ACTION TEST_CASE_2_EXEC:
                        IF vTestCases[1].state = utTestCaseStates.ut_RUNNING THEN
	(*Run the test case*)
	IF NOT assertNotEqual_STRING(vTestCase2_act, vTestCase2_xp) THEN
		vTestCases[1].state := utTestCaseStates.ut_PASSED;
		vTestCases[1].msg := 'Passed parameters were equal and function returned FALSE -> PASS';
	ELSE
		vTestCases[1].state := utTestCaseStates.ut_FAILED;
		vTestCases[1].msg := 'Passed parameters were equal and function returned TRUE -> FAIL';
	END_IF
END_IF
                      
END_ACTION
END_PROGRAM

PROGRAM test_assertNotEqual_TIME_OF_DAY
  VAR
    vTestCases : ARRAY[0..20] OF utTestCase;  (* Definition of all test cases for this POU *)
    testRunner : utTestSuite;  (* Test Suite fb instance to run the tests *)
    vRunAll : BOOL;  (* Manual command to run all tests for this POU *)
    vResetAll : BOOL;  (* Manual command to reset all tests for this POU *)
    vTestCase1_act : TOD;  (* Test data 1 of test case 1 *)
    vTestCase1_xp : TOD;  (* Test data 2 of test case 1 *)
    vTestCase2_act : TOD;  (* Test data 1 of test case 2 *)
    vTestCase2_xp : TOD;  (* Test data 2 of test case 2 *)
  END_VAR

                    (*Run the test cases*)
TEST_CASE_1_SETUP();
TEST_CASE_1_EXEC();

TEST_CASE_2_SETUP();
TEST_CASE_2_EXEC();

(*Instantiate the test runner*)
testRunner(
	Id := 48,
	Name := 'assertNotEqual_TIME_OF_DAY',
    RunTests := GVL.RunAll OR vRunAll,
	ResetTests := GVL.ResetAll OR vResetAll,
	TestCases:=vTestCases);

(*Report the results to the collection global*)
GVL.Results[testRunner.Id] := testRunner.Summary;
                  

ACTION TEST_CASE_2_EXEC:
                        IF vTestCases[1].state = utTestCaseStates.ut_RUNNING THEN
	(*Run the test case*)
	IF NOT assertNotEqual_TIME_OF_DAY(vTestCase2_act, vTestCase2_xp) THEN
		vTestCases[1].state := utTestCaseStates.ut_PASSED;
		vTestCases[1].msg := 'Passed parameters were equal and function returned FALSE -> PASS';
	ELSE
		vTestCases[1].state := utTestCaseStates.ut_FAILED;
		vTestCases[1].msg := 'Passed parameters were equal and function returned TRUE -> FAIL';
	END_IF
END_IF
                      
END_ACTION

ACTION TEST_CASE_1_SETUP:
                        IF vTestCases[0].state = utTestCaseStates.ut_SETUP THEN
	(*Setup the test case information*)
	vTestCases[0].id := 1;
	vTestCases[0].desc[0] := 'RETURNS TRUE WHEN PARAMETERS NOT EQUAL';
    vTestCases[0].desc[1] := 'Tests if the function returns True if the passed in parameters do not hold the same value';
	vTestCases[0].desc[2] := 'PASS IF: Return value is TRUE';
	
	(*Setup needed variables*)
	vTestCase1_act := REAL_TO_TOD(115.4);
	vTestCase1_xp := REAL_TO_TOD(-85.4);
END_IF
                      
END_ACTION

ACTION TEST_CASE_1_EXEC:
                        IF vTestCases[0].state = utTestCaseStates.ut_RUNNING THEN
	(*Run the test case*)
	IF assertNotEqual_TIME_OF_DAY(vTestCase1_act, vTestCase1_xp) THEN
		vTestCases[0].state := utTestCaseStates.ut_PASSED;
		vTestCases[0].msg := 'Passed parameters were not equal and function returned TRUE -> PASS';
	ELSE
		vTestCases[0].state := utTestCaseStates.ut_FAILED;
		vTestCases[0].msg := 'Passed parameters were not equal and function returned FALSE -> FAIL';
	END_IF
END_IF
                      
END_ACTION

ACTION TEST_CASE_2_SETUP:
                        IF vTestCases[1].state = utTestCaseStates.ut_SETUP THEN
	(*Setup the test case information*)
	vTestCases[1].id := 2;
	vTestCases[1].desc[0] := 'RETURNS FALSE WHEN PARAMETERS EQUAL';
    vTestCases[1].desc[1] := 'Tests if the function returns False if the passed in parameters hold the same value';
	vTestCases[1].desc[2] := 'PASS IF: Return value is FALSE';
	
	(*Setup needed variables*)
	vTestCase2_act := REAL_TO_TOD(115.4);
	vTestCase2_xp := REAL_TO_TOD(115.4);
END_IF
                      
END_ACTION
END_PROGRAM

PROGRAM test_assertGreater_UDINT
  VAR
    vTestCases : ARRAY[0..20] OF utTestCase;  (* Definition of all test cases for this POU *)
    testRunner : utTestSuite;  (* Test Suite fb instance to run the tests *)
    vRunAll : BOOL;  (* Manual command to run all tests for this POU *)
    vResetAll : BOOL;  (* Manual command to reset all tests for this POU *)
    vTestCase1_act : UDINT;  (* Test data 1 of test case 1 *)
    vTestCase1_xp : UDINT;  (* Test data 2 of test case 1 *)
    vTestCase2_act : UDINT;  (* Test data 1 of test case 2 *)
    vTestCase2_xp : UDINT;  (* Test data 2 of test case 2 *)
  END_VAR

                    (*Run the test cases*)
TEST_CASE_1_SETUP();
TEST_CASE_1_EXEC();

TEST_CASE_2_SETUP();
TEST_CASE_2_EXEC();

(*Instantiate the test runner*)
testRunner(
	Id := 59,
	Name := 'assertGreater_UDINT',
    RunTests := GVL.RunAll OR vRunAll,
	ResetTests := GVL.ResetAll OR vResetAll,
	TestCases:=vTestCases);

(*Report the results to the collection global*)
GVL.Results[testRunner.Id] := testRunner.Summary;
                  

ACTION TEST_CASE_1_SETUP:
                        IF vTestCases[0].state = utTestCaseStates.ut_SETUP THEN
	(*Setup the test case information*)
	vTestCases[0].id := 1;
	vTestCases[0].desc[0] := 'RETURNS TRUE WHEN PARAMETER ACT GREATER THAN XP';
    vTestCases[0].desc[1] := 'Tests if the function returns True if the parameter act is greater than parameter xp';
	vTestCases[0].desc[2] := 'PASS IF: Return value is TRUE';
	
	(*Setup needed variables*)
	vTestCase1_act := REAL_TO_UDINT(115.4);
	vTestCase1_xp := REAL_TO_UDINT(85.4);
END_IF
                      
END_ACTION

ACTION TEST_CASE_1_EXEC:
                        IF vTestCases[0].state = utTestCaseStates.ut_RUNNING THEN
	(*Run the test case*)
	IF assertGreater_UDINT(vTestCase1_act, vTestCase1_xp) THEN
		vTestCases[0].state := utTestCaseStates.ut_PASSED;
		vTestCases[0].msg := 'Parameter act was greater than xp and function returned TRUE -> PASS';
	ELSE
		vTestCases[0].state := utTestCaseStates.ut_FAILED;
		vTestCases[0].msg := 'Parameter act was greater than xp and function returned FALSE -> FAIL';
	END_IF
END_IF
                      
END_ACTION

ACTION TEST_CASE_2_SETUP:
                        IF vTestCases[1].state = utTestCaseStates.ut_SETUP THEN
	(*Setup the test case information*)
	vTestCases[1].id := 2;
    vTestCases[1].desc[0] := 'RETURNS FALSE WHEN PARAMETER ACT LESS THAN XP';
    vTestCases[1].desc[1] := 'Tests if the function returns False if the parameter act is less than parameter xp';
	vTestCases[1].desc[2] := 'PASS IF: Return value is FALSE';
	
	(*Setup needed variables*)
	vTestCase2_act := REAL_TO_UDINT(8.4);
	vTestCase2_xp := REAL_TO_UDINT(85.4);
END_IF
                      
END_ACTION

ACTION TEST_CASE_2_EXEC:
                        IF vTestCases[1].state = utTestCaseStates.ut_RUNNING THEN
	(*Run the test case*)
	IF NOT assertGreater_UDINT(vTestCase2_act, vTestCase2_xp) THEN
		vTestCases[1].state := utTestCaseStates.ut_PASSED;
		vTestCases[1].msg := 'Parameter act was less than xp and function returned FALSE -> PASS';
	ELSE
		vTestCases[1].state := utTestCaseStates.ut_FAILED;
		vTestCases[1].msg := 'Parameter act was less than xp and function returned TRUE -> FAIL';
	END_IF
END_IF
                      
END_ACTION
END_PROGRAM

PROGRAM test_assertNotEqual_LTIME_OF_DAY
  VAR
    vTestCases : ARRAY[0..20] OF utTestCase;  (* Definition of all test cases for this POU *)
    testRunner : utTestSuite;  (* Test Suite fb instance to run the tests *)
    vRunAll : BOOL;  (* Manual command to run all tests for this POU *)
    vResetAll : BOOL;  (* Manual command to reset all tests for this POU *)
    vTestCase1_act : LTIME_OF_DAY;  (* Test data 1 of test case 1 *)
    vTestCase1_xp : LTIME_OF_DAY;  (* Test data 2 of test case 1 *)
    vTestCase2_act : LTIME_OF_DAY;  (* Test data 1 of test case 2 *)
    vTestCase2_xp : LTIME_OF_DAY;  (* Test data 2 of test case 2 *)
  END_VAR

                    (*Run the test cases*)
TEST_CASE_1_SETUP();
TEST_CASE_1_EXEC();

TEST_CASE_2_SETUP();
TEST_CASE_2_EXEC();

(*Instantiate the test runner*)
testRunner(
	Id := 49,
	Name := 'assertNotEqual_LTIME_OF_DAY',
    RunTests := GVL.RunAll OR vRunAll,
	ResetTests := GVL.ResetAll OR vResetAll,
	TestCases:=vTestCases);

(*Report the results to the collection global*)
GVL.Results[testRunner.Id] := testRunner.Summary;
                  

ACTION TEST_CASE_1_SETUP:
                        IF vTestCases[0].state = utTestCaseStates.ut_SETUP THEN
	(*Setup the test case information*)
	vTestCases[0].id := 1;
	vTestCases[0].desc[0] := 'RETURNS TRUE WHEN PARAMETERS NOT EQUAL';
    vTestCases[0].desc[1] := 'Tests if the function returns True if the passed in parameters do not hold the same value';
	vTestCases[0].desc[2] := 'PASS IF: Return value is TRUE';
	
	(*Setup needed variables*)
	vTestCase1_act := REAL_TO_LTOD(115.4);
	vTestCase1_xp := REAL_TO_LTOD(-85.4);
END_IF
                      
END_ACTION

ACTION TEST_CASE_1_EXEC:
                        IF vTestCases[0].state = utTestCaseStates.ut_RUNNING THEN
	(*Run the test case*)
	IF assertNotEqual_LTIME_OF_DAY(vTestCase1_act, vTestCase1_xp) THEN
		vTestCases[0].state := utTestCaseStates.ut_PASSED;
		vTestCases[0].msg := 'Passed parameters were not equal and function returned TRUE -> PASS';
	ELSE
		vTestCases[0].state := utTestCaseStates.ut_FAILED;
		vTestCases[0].msg := 'Passed parameters were not equal and function returned FALSE -> FAIL';
	END_IF
END_IF
                      
END_ACTION

ACTION TEST_CASE_2_SETUP:
                        IF vTestCases[1].state = utTestCaseStates.ut_SETUP THEN
	(*Setup the test case information*)
	vTestCases[1].id := 2;
	vTestCases[1].desc[0] := 'RETURNS FALSE WHEN PARAMETERS EQUAL';
    vTestCases[1].desc[1] := 'Tests if the function returns False if the passed in parameters hold the same value';
	vTestCases[1].desc[2] := 'PASS IF: Return value is FALSE';
	
	(*Setup needed variables*)
	vTestCase2_act := REAL_TO_LTOD(115.4);
	vTestCase2_xp := REAL_TO_LTOD(115.4);
END_IF
                      
END_ACTION

ACTION TEST_CASE_2_EXEC:
                        IF vTestCases[1].state = utTestCaseStates.ut_RUNNING THEN
	(*Run the test case*)
	IF NOT assertNotEqual_LTIME_OF_DAY(vTestCase2_act, vTestCase2_xp) THEN
		vTestCases[1].state := utTestCaseStates.ut_PASSED;
		vTestCases[1].msg := 'Passed parameters were equal and function returned FALSE -> PASS';
	ELSE
		vTestCases[1].state := utTestCaseStates.ut_FAILED;
		vTestCases[1].msg := 'Passed parameters were equal and function returned TRUE -> FAIL';
	END_IF
END_IF
                      
END_ACTION
END_PROGRAM

PROGRAM test_assertGreater_BYTE
  VAR
    vTestCases : ARRAY[0..20] OF utTestCase;  (* Definition of all test cases for this POU *)
    testRunner : utTestSuite;  (* Test Suite fb instance to run the tests *)
    vRunAll : BOOL;  (* Manual command to run all tests for this POU *)
    vResetAll : BOOL;  (* Manual command to reset all tests for this POU *)
    vTestCase1_act : BYTE;  (* Test data 1 of test case 1 *)
    vTestCase1_xp : BYTE;  (* Test data 2 of test case 1 *)
    vTestCase2_act : BYTE;  (* Test data 1 of test case 2 *)
    vTestCase2_xp : BYTE;  (* Test data 2 of test case 2 *)
  END_VAR

                    (*Run the test cases*)
TEST_CASE_1_SETUP();
TEST_CASE_1_EXEC();

TEST_CASE_2_SETUP();
TEST_CASE_2_EXEC();

(*Instantiate the test runner*)
testRunner(
	Id := 50,
	Name := 'assertGreater_BYTE',
    RunTests := GVL.RunAll OR vRunAll,
	ResetTests := GVL.ResetAll OR vResetAll,
	TestCases:=vTestCases);

(*Report the results to the collection global*)
GVL.Results[testRunner.Id] := testRunner.Summary;
                  

ACTION TEST_CASE_1_SETUP:
                        IF vTestCases[0].state = utTestCaseStates.ut_SETUP THEN
	(*Setup the test case information*)
	vTestCases[0].id := 1;
	vTestCases[0].desc[0] := 'RETURNS TRUE WHEN PARAMETER ACT GREATER THAN XP';
    vTestCases[0].desc[1] := 'Tests if the function returns True if the parameter act is greater than parameter xp';
	vTestCases[0].desc[2] := 'PASS IF: Return value is TRUE';
	
	(*Setup needed variables*)
	vTestCase1_act := REAL_TO_BYTE(115.4);
	vTestCase1_xp := REAL_TO_BYTE(85.4);
END_IF
                      
END_ACTION

ACTION TEST_CASE_1_EXEC:
                        IF vTestCases[0].state = utTestCaseStates.ut_RUNNING THEN
	(*Run the test case*)
	IF assertGreater_BYTE(vTestCase1_act, vTestCase1_xp) THEN
		vTestCases[0].state := utTestCaseStates.ut_PASSED;
		vTestCases[0].msg := 'Parameter act was greater than xp and function returned TRUE -> PASS';
	ELSE
		vTestCases[0].state := utTestCaseStates.ut_FAILED;
		vTestCases[0].msg := 'Parameter act was greater than xp and function returned FALSE -> FAIL';
	END_IF
END_IF
                      
END_ACTION

ACTION TEST_CASE_2_SETUP:
                        IF vTestCases[1].state = utTestCaseStates.ut_SETUP THEN
	(*Setup the test case information*)
	vTestCases[1].id := 2;
    vTestCases[1].desc[0] := 'RETURNS FALSE WHEN PARAMETER ACT LESS THAN XP';
    vTestCases[1].desc[1] := 'Tests if the function returns False if the parameter act is less than parameter xp';
	vTestCases[1].desc[2] := 'PASS IF: Return value is FALSE';
	
	(*Setup needed variables*)
	vTestCase2_act := REAL_TO_BYTE(8.4);
	vTestCase2_xp := REAL_TO_BYTE(85.4);
END_IF
                      
END_ACTION

ACTION TEST_CASE_2_EXEC:
                        IF vTestCases[1].state = utTestCaseStates.ut_RUNNING THEN
	(*Run the test case*)
	IF NOT assertGreater_BYTE(vTestCase2_act, vTestCase2_xp) THEN
		vTestCases[1].state := utTestCaseStates.ut_PASSED;
		vTestCases[1].msg := 'Parameter act was less than xp and function returned FALSE -> PASS';
	ELSE
		vTestCases[1].state := utTestCaseStates.ut_FAILED;
		vTestCases[1].msg := 'Parameter act was less than xp and function returned TRUE -> FAIL';
	END_IF
END_IF
                      
END_ACTION
END_PROGRAM

PROGRAM test_assertNotEqual_WSTRING
  VAR
    vTestCases : ARRAY[0..20] OF utTestCase;  (* Definition of all test cases for this POU *)
    testRunner : utTestSuite;  (* Test Suite fb instance to run the tests *)
    vRunAll : BOOL;  (* Manual command to run all tests for this POU *)
    vResetAll : BOOL;  (* Manual command to reset all tests for this POU *)
    vTestCase1_act : WSTRING;  (* Test data 1 of test case 1 *)
    vTestCase1_xp : WSTRING;  (* Test data 2 of test case 1 *)
    vTestCase2_act : WSTRING;  (* Test data 1 of test case 2 *)
    vTestCase2_xp : WSTRING;  (* Test data 2 of test case 2 *)
  END_VAR

                    (*Run the test cases*)
TEST_CASE_1_SETUP();
TEST_CASE_1_EXEC();

TEST_CASE_2_SETUP();
TEST_CASE_2_EXEC();

(*Instantiate the test runner*)
testRunner(
	Id := 41,
	Name := 'assertNotEqual_WSTRING',
    RunTests := GVL.RunAll OR vRunAll,
	ResetTests := GVL.ResetAll OR vResetAll,
	TestCases:=vTestCases);

(*Report the results to the collection global*)
GVL.Results[testRunner.Id] := testRunner.Summary;
                  

ACTION TEST_CASE_2_EXEC:
                        IF vTestCases[1].state = utTestCaseStates.ut_RUNNING THEN
	(*Run the test case*)
	IF NOT assertNotEqual_WSTRING(vTestCase2_act, vTestCase2_xp) THEN
		vTestCases[1].state := utTestCaseStates.ut_PASSED;
		vTestCases[1].msg := 'Passed parameters were equal and function returned FALSE -> PASS';
	ELSE
		vTestCases[1].state := utTestCaseStates.ut_FAILED;
		vTestCases[1].msg := 'Passed parameters were equal and function returned TRUE -> FAIL';
	END_IF
END_IF
                      
END_ACTION

ACTION TEST_CASE_1_SETUP:
                        IF vTestCases[0].state = utTestCaseStates.ut_SETUP THEN
	(*Setup the test case information*)
	vTestCases[0].id := 1;
	vTestCases[0].desc[0] := 'RETURNS TRUE WHEN PARAMETERS NOT EQUAL';
    vTestCases[0].desc[1] := 'Tests if the function returns True if the passed in parameters do not hold the same value';
	vTestCases[0].desc[2] := 'PASS IF: Return value is TRUE';
	
	(*Setup needed variables*)
	vTestCase1_act := REAL_TO_WSTRING(115.4);
	vTestCase1_xp := REAL_TO_WSTRING(-85.4);
END_IF
                      
END_ACTION

ACTION TEST_CASE_1_EXEC:
                        IF vTestCases[0].state = utTestCaseStates.ut_RUNNING THEN
	(*Run the test case*)
	IF assertNotEqual_WSTRING(vTestCase1_act, vTestCase1_xp) THEN
		vTestCases[0].state := utTestCaseStates.ut_PASSED;
		vTestCases[0].msg := 'Passed parameters were not equal and function returned TRUE -> PASS';
	ELSE
		vTestCases[0].state := utTestCaseStates.ut_FAILED;
		vTestCases[0].msg := 'Passed parameters were not equal and function returned FALSE -> FAIL';
	END_IF
END_IF
                      
END_ACTION

ACTION TEST_CASE_2_SETUP:
                        IF vTestCases[1].state = utTestCaseStates.ut_SETUP THEN
	(*Setup the test case information*)
	vTestCases[1].id := 2;
	vTestCases[1].desc[0] := 'RETURNS FALSE WHEN PARAMETERS EQUAL';
    vTestCases[1].desc[1] := 'Tests if the function returns False if the passed in parameters hold the same value';
	vTestCases[1].desc[2] := 'PASS IF: Return value is FALSE';
	
	(*Setup needed variables*)
	vTestCase2_act := REAL_TO_WSTRING(115.4);
	vTestCase2_xp := REAL_TO_WSTRING(115.4);
END_IF
                      
END_ACTION
END_PROGRAM

PROGRAM test_assertNotEqual_DWORD
  VAR
    vTestCases : ARRAY[0..20] OF utTestCase;  (* Definition of all test cases for this POU *)
    testRunner : utTestSuite;  (* Test Suite fb instance to run the tests *)
    vRunAll : BOOL;  (* Manual command to run all tests for this POU *)
    vResetAll : BOOL;  (* Manual command to reset all tests for this POU *)
    vTestCase1_act : DWORD;  (* Test data 1 of test case 1 *)
    vTestCase1_xp : DWORD;  (* Test data 2 of test case 1 *)
    vTestCase2_act : DWORD;  (* Test data 1 of test case 2 *)
    vTestCase2_xp : DWORD;  (* Test data 2 of test case 2 *)
  END_VAR

                    (*Run the test cases*)
TEST_CASE_1_SETUP();
TEST_CASE_1_EXEC();

TEST_CASE_2_SETUP();
TEST_CASE_2_EXEC();

(*Instantiate the test runner*)
testRunner(
	Id := 28,
	Name := 'assertNotEqual_DWORD',
    RunTests := GVL.RunAll OR vRunAll,
	ResetTests := GVL.ResetAll OR vResetAll,
	TestCases:=vTestCases);

(*Report the results to the collection global*)
GVL.Results[testRunner.Id] := testRunner.Summary;
                  

ACTION TEST_CASE_1_SETUP:
                        IF vTestCases[0].state = utTestCaseStates.ut_SETUP THEN
	(*Setup the test case information*)
	vTestCases[0].id := 1;
	vTestCases[0].desc[0] := 'RETURNS TRUE WHEN PARAMETERS NOT EQUAL';
    vTestCases[0].desc[1] := 'Tests if the function returns True if the passed in parameters do not hold the same value';
	vTestCases[0].desc[2] := 'PASS IF: Return value is TRUE';
	
	(*Setup needed variables*)
	vTestCase1_act := REAL_TO_DWORD(115.4);
	vTestCase1_xp := REAL_TO_DWORD(-85.4);
END_IF
                      
END_ACTION

ACTION TEST_CASE_1_EXEC:
                        IF vTestCases[0].state = utTestCaseStates.ut_RUNNING THEN
	(*Run the test case*)
	IF assertNotEqual_DWORD(vTestCase1_act, vTestCase1_xp) THEN
		vTestCases[0].state := utTestCaseStates.ut_PASSED;
		vTestCases[0].msg := 'Passed parameters were not equal and function returned TRUE -> PASS';
	ELSE
		vTestCases[0].state := utTestCaseStates.ut_FAILED;
		vTestCases[0].msg := 'Passed parameters were not equal and function returned FALSE -> FAIL';
	END_IF
END_IF
                      
END_ACTION

ACTION TEST_CASE_2_SETUP:
                        IF vTestCases[1].state = utTestCaseStates.ut_SETUP THEN
	(*Setup the test case information*)
	vTestCases[1].id := 2;
	vTestCases[1].desc[0] := 'RETURNS FALSE WHEN PARAMETERS EQUAL';
    vTestCases[1].desc[1] := 'Tests if the function returns False if the passed in parameters hold the same value';
	vTestCases[1].desc[2] := 'PASS IF: Return value is FALSE';
	
	(*Setup needed variables*)
	vTestCase2_act := REAL_TO_DWORD(115.4);
	vTestCase2_xp := REAL_TO_DWORD(115.4);
END_IF
                      
END_ACTION

ACTION TEST_CASE_2_EXEC:
                        IF vTestCases[1].state = utTestCaseStates.ut_RUNNING THEN
	(*Run the test case*)
	IF NOT assertNotEqual_DWORD(vTestCase2_act, vTestCase2_xp) THEN
		vTestCases[1].state := utTestCaseStates.ut_PASSED;
		vTestCases[1].msg := 'Passed parameters were equal and function returned FALSE -> PASS';
	ELSE
		vTestCases[1].state := utTestCaseStates.ut_FAILED;
		vTestCases[1].msg := 'Passed parameters were equal and function returned TRUE -> FAIL';
	END_IF
END_IF
                      
END_ACTION
END_PROGRAM

PROGRAM test_assertNotEqual_LWORD
  VAR
    vTestCases : ARRAY[0..20] OF utTestCase;  (* Definition of all test cases for this POU *)
    testRunner : utTestSuite;  (* Test Suite fb instance to run the tests *)
    vRunAll : BOOL;  (* Manual command to run all tests for this POU *)
    vResetAll : BOOL;  (* Manual command to reset all tests for this POU *)
    vTestCase1_act : LWORD;  (* Test data 1 of test case 1 *)
    vTestCase1_xp : LWORD;  (* Test data 2 of test case 1 *)
    vTestCase2_act : LWORD;  (* Test data 1 of test case 2 *)
    vTestCase2_xp : LWORD;  (* Test data 2 of test case 2 *)
  END_VAR

                    (*Run the test cases*)
TEST_CASE_1_SETUP();
TEST_CASE_1_EXEC();

TEST_CASE_2_SETUP();
TEST_CASE_2_EXEC();

(*Instantiate the test runner*)
testRunner(
	Id := 29,
	Name := 'assertNotEqual_LWORD',
    RunTests := GVL.RunAll OR vRunAll,
	ResetTests := GVL.ResetAll OR vResetAll,
	TestCases:=vTestCases);

(*Report the results to the collection global*)
GVL.Results[testRunner.Id] := testRunner.Summary;
                  

ACTION TEST_CASE_1_SETUP:
                        IF vTestCases[0].state = utTestCaseStates.ut_SETUP THEN
	(*Setup the test case information*)
	vTestCases[0].id := 1;
	vTestCases[0].desc[0] := 'RETURNS TRUE WHEN PARAMETERS NOT EQUAL';
    vTestCases[0].desc[1] := 'Tests if the function returns True if the passed in parameters do not hold the same value';
	vTestCases[0].desc[2] := 'PASS IF: Return value is TRUE';
	
	(*Setup needed variables*)
	vTestCase1_act := REAL_TO_LWORD(115.4);
	vTestCase1_xp := REAL_TO_LWORD(-85.4);
END_IF
                      
END_ACTION

ACTION TEST_CASE_1_EXEC:
                        IF vTestCases[0].state = utTestCaseStates.ut_RUNNING THEN
	(*Run the test case*)
	IF assertNotEqual_LWORD(vTestCase1_act, vTestCase1_xp) THEN
		vTestCases[0].state := utTestCaseStates.ut_PASSED;
		vTestCases[0].msg := 'Passed parameters were not equal and function returned TRUE -> PASS';
	ELSE
		vTestCases[0].state := utTestCaseStates.ut_FAILED;
		vTestCases[0].msg := 'Passed parameters were not equal and function returned FALSE -> FAIL';
	END_IF
END_IF
                      
END_ACTION

ACTION TEST_CASE_2_SETUP:
                        IF vTestCases[1].state = utTestCaseStates.ut_SETUP THEN
	(*Setup the test case information*)
	vTestCases[1].id := 2;
	vTestCases[1].desc[0] := 'RETURNS FALSE WHEN PARAMETERS EQUAL';
    vTestCases[1].desc[1] := 'Tests if the function returns False if the passed in parameters hold the same value';
	vTestCases[1].desc[2] := 'PASS IF: Return value is FALSE';
	
	(*Setup needed variables*)
	vTestCase2_act := REAL_TO_LWORD(115.4);
	vTestCase2_xp := REAL_TO_LWORD(115.4);
END_IF
                      
END_ACTION

ACTION TEST_CASE_2_EXEC:
                        IF vTestCases[1].state = utTestCaseStates.ut_RUNNING THEN
	(*Run the test case*)
	IF NOT assertNotEqual_LWORD(vTestCase2_act, vTestCase2_xp) THEN
		vTestCases[1].state := utTestCaseStates.ut_PASSED;
		vTestCases[1].msg := 'Passed parameters were equal and function returned FALSE -> PASS';
	ELSE
		vTestCases[1].state := utTestCaseStates.ut_FAILED;
		vTestCases[1].msg := 'Passed parameters were equal and function returned TRUE -> FAIL';
	END_IF
END_IF
                      
END_ACTION
END_PROGRAM

PROGRAM test_assertNotEqual_UDINT
  VAR
    vTestCases : ARRAY[0..20] OF utTestCase;  (* Definition of all test cases for this POU *)
    testRunner : utTestSuite;  (* Test Suite fb instance to run the tests *)
    vRunAll : BOOL;  (* Manual command to run all tests for this POU *)
    vResetAll : BOOL;  (* Manual command to reset all tests for this POU *)
    vTestCase1_act : UDINT;  (* Test data 1 of test case 1 *)
    vTestCase1_xp : UDINT;  (* Test data 2 of test case 1 *)
    vTestCase2_act : UDINT;  (* Test data 1 of test case 2 *)
    vTestCase2_xp : UDINT;  (* Test data 2 of test case 2 *)
  END_VAR

                    (*Run the test cases*)
TEST_CASE_1_SETUP();
TEST_CASE_1_EXEC();

TEST_CASE_2_SETUP();
TEST_CASE_2_EXEC();

(*Instantiate the test runner*)
testRunner(
	Id := 35,
	Name := 'assertNotEqual_UDINT',
    RunTests := GVL.RunAll OR vRunAll,
	ResetTests := GVL.ResetAll OR vResetAll,
	TestCases:=vTestCases);

(*Report the results to the collection global*)
GVL.Results[testRunner.Id] := testRunner.Summary;
                  

ACTION TEST_CASE_1_SETUP:
                        IF vTestCases[0].state = utTestCaseStates.ut_SETUP THEN
	(*Setup the test case information*)
	vTestCases[0].id := 1;
	vTestCases[0].desc[0] := 'RETURNS TRUE WHEN PARAMETERS NOT EQUAL';
    vTestCases[0].desc[1] := 'Tests if the function returns True if the passed in parameters do not hold the same value';
	vTestCases[0].desc[2] := 'PASS IF: Return value is TRUE';
	
	(*Setup needed variables*)
	vTestCase1_act := REAL_TO_UDINT(115.4);
	vTestCase1_xp := REAL_TO_UDINT(-85.4);
END_IF
                      
END_ACTION

ACTION TEST_CASE_1_EXEC:
                        IF vTestCases[0].state = utTestCaseStates.ut_RUNNING THEN
	(*Run the test case*)
	IF assertNotEqual_UDINT(vTestCase1_act, vTestCase1_xp) THEN
		vTestCases[0].state := utTestCaseStates.ut_PASSED;
		vTestCases[0].msg := 'Passed parameters were not equal and function returned TRUE -> PASS';
	ELSE
		vTestCases[0].state := utTestCaseStates.ut_FAILED;
		vTestCases[0].msg := 'Passed parameters were not equal and function returned FALSE -> FAIL';
	END_IF
END_IF
                      
END_ACTION

ACTION TEST_CASE_2_SETUP:
                        IF vTestCases[1].state = utTestCaseStates.ut_SETUP THEN
	(*Setup the test case information*)
	vTestCases[1].id := 2;
	vTestCases[1].desc[0] := 'RETURNS FALSE WHEN PARAMETERS EQUAL';
    vTestCases[1].desc[1] := 'Tests if the function returns False if the passed in parameters hold the same value';
	vTestCases[1].desc[2] := 'PASS IF: Return value is FALSE';
	
	(*Setup needed variables*)
	vTestCase2_act := REAL_TO_UDINT(115.4);
	vTestCase2_xp := REAL_TO_UDINT(115.4);
END_IF
                      
END_ACTION

ACTION TEST_CASE_2_EXEC:
                        IF vTestCases[1].state = utTestCaseStates.ut_RUNNING THEN
	(*Run the test case*)
	IF NOT assertNotEqual_UDINT(vTestCase2_act, vTestCase2_xp) THEN
		vTestCases[1].state := utTestCaseStates.ut_PASSED;
		vTestCases[1].msg := 'Passed parameters were equal and function returned FALSE -> PASS';
	ELSE
		vTestCases[1].state := utTestCaseStates.ut_FAILED;
		vTestCases[1].msg := 'Passed parameters were equal and function returned TRUE -> FAIL';
	END_IF
END_IF
                      
END_ACTION
END_PROGRAM

PROGRAM test_assertNotEqual_LINT
  VAR
    vTestCases : ARRAY[0..20] OF utTestCase;  (* Definition of all test cases for this POU *)
    testRunner : utTestSuite;  (* Test Suite fb instance to run the tests *)
    vRunAll : BOOL;  (* Manual command to run all tests for this POU *)
    vResetAll : BOOL;  (* Manual command to reset all tests for this POU *)
    vTestCase1_act : LINT;  (* Test data 1 of test case 1 *)
    vTestCase1_xp : LINT;  (* Test data 2 of test case 1 *)
    vTestCase2_act : LINT;  (* Test data 1 of test case 2 *)
    vTestCase2_xp : LINT;  (* Test data 2 of test case 2 *)
  END_VAR

                    (*Run the test cases*)
TEST_CASE_1_SETUP();
TEST_CASE_1_EXEC();

TEST_CASE_2_SETUP();
TEST_CASE_2_EXEC();

(*Instantiate the test runner*)
testRunner(
	Id := 36,
	Name := 'assertNotEqual_LINT',
    RunTests := GVL.RunAll OR vRunAll,
	ResetTests := GVL.ResetAll OR vResetAll,
	TestCases:=vTestCases);

(*Report the results to the collection global*)
GVL.Results[testRunner.Id] := testRunner.Summary;
                  

ACTION TEST_CASE_1_SETUP:
                        IF vTestCases[0].state = utTestCaseStates.ut_SETUP THEN
	(*Setup the test case information*)
	vTestCases[0].id := 1;
	vTestCases[0].desc[0] := 'RETURNS TRUE WHEN PARAMETERS NOT EQUAL';
    vTestCases[0].desc[1] := 'Tests if the function returns True if the passed in parameters do not hold the same value';
	vTestCases[0].desc[2] := 'PASS IF: Return value is TRUE';
	
	(*Setup needed variables*)
	vTestCase1_act := REAL_TO_LINT(115.4);
	vTestCase1_xp := REAL_TO_LINT(-85.4);
END_IF
                      
END_ACTION

ACTION TEST_CASE_1_EXEC:
                        IF vTestCases[0].state = utTestCaseStates.ut_RUNNING THEN
	(*Run the test case*)
	IF assertNotEqual_LINT(vTestCase1_act, vTestCase1_xp) THEN
		vTestCases[0].state := utTestCaseStates.ut_PASSED;
		vTestCases[0].msg := 'Passed parameters were not equal and function returned TRUE -> PASS';
	ELSE
		vTestCases[0].state := utTestCaseStates.ut_FAILED;
		vTestCases[0].msg := 'Passed parameters were not equal and function returned FALSE -> FAIL';
	END_IF
END_IF
                      
END_ACTION

ACTION TEST_CASE_2_SETUP:
                        IF vTestCases[1].state = utTestCaseStates.ut_SETUP THEN
	(*Setup the test case information*)
	vTestCases[1].id := 2;
	vTestCases[1].desc[0] := 'RETURNS FALSE WHEN PARAMETERS EQUAL';
    vTestCases[1].desc[1] := 'Tests if the function returns False if the passed in parameters hold the same value';
	vTestCases[1].desc[2] := 'PASS IF: Return value is FALSE';
	
	(*Setup needed variables*)
	vTestCase2_act := REAL_TO_LINT(115.4);
	vTestCase2_xp := REAL_TO_LINT(115.4);
END_IF
                      
END_ACTION

ACTION TEST_CASE_2_EXEC:
                        IF vTestCases[1].state = utTestCaseStates.ut_RUNNING THEN
	(*Run the test case*)
	IF NOT assertNotEqual_LINT(vTestCase2_act, vTestCase2_xp) THEN
		vTestCases[1].state := utTestCaseStates.ut_PASSED;
		vTestCases[1].msg := 'Passed parameters were equal and function returned FALSE -> PASS';
	ELSE
		vTestCases[1].state := utTestCaseStates.ut_FAILED;
		vTestCases[1].msg := 'Passed parameters were equal and function returned TRUE -> FAIL';
	END_IF
END_IF
                      
END_ACTION
END_PROGRAM

PROGRAM test_assertNotEqual_SINT
  VAR
    vTestCases : ARRAY[0..20] OF utTestCase;  (* Definition of all test cases for this POU *)
    testRunner : utTestSuite;  (* Test Suite fb instance to run the tests *)
    vRunAll : BOOL;  (* Manual command to run all tests for this POU *)
    vResetAll : BOOL;  (* Manual command to reset all tests for this POU *)
    vTestCase1_act : SINT;  (* Test data 1 of test case 1 *)
    vTestCase1_xp : SINT;  (* Test data 2 of test case 1 *)
    vTestCase2_act : SINT;  (* Test data 1 of test case 2 *)
    vTestCase2_xp : SINT;  (* Test data 2 of test case 2 *)
  END_VAR

                    (*Run the test cases*)
TEST_CASE_1_SETUP();
TEST_CASE_1_EXEC();

TEST_CASE_2_SETUP();
TEST_CASE_2_EXEC();

(*Instantiate the test runner*)
testRunner(
	Id := 30,
	Name := 'assertNotEqual_SINT',
    RunTests := GVL.RunAll OR vRunAll,
	ResetTests := GVL.ResetAll OR vResetAll,
	TestCases:=vTestCases);

(*Report the results to the collection global*)
GVL.Results[testRunner.Id] := testRunner.Summary;
                  

ACTION TEST_CASE_2_SETUP:
                        IF vTestCases[1].state = utTestCaseStates.ut_SETUP THEN
	(*Setup the test case information*)
	vTestCases[1].id := 2;
	vTestCases[1].desc[0] := 'RETURNS FALSE WHEN PARAMETERS EQUAL';
    vTestCases[1].desc[1] := 'Tests if the function returns False if the passed in parameters hold the same value';
	vTestCases[1].desc[2] := 'PASS IF: Return value is FALSE';
	
	(*Setup needed variables*)
	vTestCase2_act := REAL_TO_SINT(115.4);
	vTestCase2_xp := REAL_TO_SINT(115.4);
END_IF
                      
END_ACTION

ACTION TEST_CASE_2_EXEC:
                        IF vTestCases[1].state = utTestCaseStates.ut_RUNNING THEN
	(*Run the test case*)
	IF NOT assertNotEqual_SINT(vTestCase2_act, vTestCase2_xp) THEN
		vTestCases[1].state := utTestCaseStates.ut_PASSED;
		vTestCases[1].msg := 'Passed parameters were equal and function returned FALSE -> PASS';
	ELSE
		vTestCases[1].state := utTestCaseStates.ut_FAILED;
		vTestCases[1].msg := 'Passed parameters were equal and function returned TRUE -> FAIL';
	END_IF
END_IF
                      
END_ACTION

ACTION TEST_CASE_1_SETUP:
                        IF vTestCases[0].state = utTestCaseStates.ut_SETUP THEN
	(*Setup the test case information*)
	vTestCases[0].id := 1;
	vTestCases[0].desc[0] := 'RETURNS TRUE WHEN PARAMETERS NOT EQUAL';
    vTestCases[0].desc[1] := 'Tests if the function returns True if the passed in parameters do not hold the same value';
	vTestCases[0].desc[2] := 'PASS IF: Return value is TRUE';
	
	(*Setup needed variables*)
	vTestCase1_act := REAL_TO_SINT(115.4);
	vTestCase1_xp := REAL_TO_SINT(-85.4);
END_IF
                      
END_ACTION

ACTION TEST_CASE_1_EXEC:
                        IF vTestCases[0].state = utTestCaseStates.ut_RUNNING THEN
	(*Run the test case*)
	IF assertNotEqual_SINT(vTestCase1_act, vTestCase1_xp) THEN
		vTestCases[0].state := utTestCaseStates.ut_PASSED;
		vTestCases[0].msg := 'Passed parameters were not equal and function returned TRUE -> PASS';
	ELSE
		vTestCases[0].state := utTestCaseStates.ut_FAILED;
		vTestCases[0].msg := 'Passed parameters were not equal and function returned FALSE -> FAIL';
	END_IF
END_IF
                      
END_ACTION
END_PROGRAM

PROGRAM test_assertNotEqual_ULINT
  VAR
    vTestCases : ARRAY[0..20] OF utTestCase;  (* Definition of all test cases for this POU *)
    testRunner : utTestSuite;  (* Test Suite fb instance to run the tests *)
    vRunAll : BOOL;  (* Manual command to run all tests for this POU *)
    vResetAll : BOOL;  (* Manual command to reset all tests for this POU *)
    vTestCase1_act : ULINT;  (* Test data 1 of test case 1 *)
    vTestCase1_xp : ULINT;  (* Test data 2 of test case 1 *)
    vTestCase2_act : ULINT;  (* Test data 1 of test case 2 *)
    vTestCase2_xp : ULINT;  (* Test data 2 of test case 2 *)
  END_VAR

                    (*Run the test cases*)
TEST_CASE_1_SETUP();
TEST_CASE_1_EXEC();

TEST_CASE_2_SETUP();
TEST_CASE_2_EXEC();

(*Instantiate the test runner*)
testRunner(
	Id := 37,
	Name := 'assertNotEqual_ULINT',
    RunTests := GVL.RunAll OR vRunAll,
	ResetTests := GVL.ResetAll OR vResetAll,
	TestCases:=vTestCases);

(*Report the results to the collection global*)
GVL.Results[testRunner.Id] := testRunner.Summary;
                  

ACTION TEST_CASE_2_SETUP:
                        IF vTestCases[1].state = utTestCaseStates.ut_SETUP THEN
	(*Setup the test case information*)
	vTestCases[1].id := 2;
	vTestCases[1].desc[0] := 'RETURNS FALSE WHEN PARAMETERS EQUAL';
    vTestCases[1].desc[1] := 'Tests if the function returns False if the passed in parameters hold the same value';
	vTestCases[1].desc[2] := 'PASS IF: Return value is FALSE';
	
	(*Setup needed variables*)
	vTestCase2_act := REAL_TO_ULINT(115.4);
	vTestCase2_xp := REAL_TO_ULINT(115.4);
END_IF
                      
END_ACTION

ACTION TEST_CASE_2_EXEC:
                        IF vTestCases[1].state = utTestCaseStates.ut_RUNNING THEN
	(*Run the test case*)
	IF NOT assertNotEqual_ULINT(vTestCase2_act, vTestCase2_xp) THEN
		vTestCases[1].state := utTestCaseStates.ut_PASSED;
		vTestCases[1].msg := 'Passed parameters were equal and function returned FALSE -> PASS';
	ELSE
		vTestCases[1].state := utTestCaseStates.ut_FAILED;
		vTestCases[1].msg := 'Passed parameters were equal and function returned TRUE -> FAIL';
	END_IF
END_IF
                      
END_ACTION

ACTION TEST_CASE_1_SETUP:
                        IF vTestCases[0].state = utTestCaseStates.ut_SETUP THEN
	(*Setup the test case information*)
	vTestCases[0].id := 1;
	vTestCases[0].desc[0] := 'RETURNS TRUE WHEN PARAMETERS NOT EQUAL';
    vTestCases[0].desc[1] := 'Tests if the function returns True if the passed in parameters do not hold the same value';
	vTestCases[0].desc[2] := 'PASS IF: Return value is TRUE';
	
	(*Setup needed variables*)
	vTestCase1_act := REAL_TO_ULINT(115.4);
	vTestCase1_xp := REAL_TO_ULINT(-85.4);
END_IF
                      
END_ACTION

ACTION TEST_CASE_1_EXEC:
                        IF vTestCases[0].state = utTestCaseStates.ut_RUNNING THEN
	(*Run the test case*)
	IF assertNotEqual_ULINT(vTestCase1_act, vTestCase1_xp) THEN
		vTestCases[0].state := utTestCaseStates.ut_PASSED;
		vTestCases[0].msg := 'Passed parameters were not equal and function returned TRUE -> PASS';
	ELSE
		vTestCases[0].state := utTestCaseStates.ut_FAILED;
		vTestCases[0].msg := 'Passed parameters were not equal and function returned FALSE -> FAIL';
	END_IF
END_IF
                      
END_ACTION
END_PROGRAM

PROGRAM test_assertGreater_WORD
  VAR
    vTestCases : ARRAY[0..20] OF utTestCase;  (* Definition of all test cases for this POU *)
    testRunner : utTestSuite;  (* Test Suite fb instance to run the tests *)
    vRunAll : BOOL;  (* Manual command to run all tests for this POU *)
    vResetAll : BOOL;  (* Manual command to reset all tests for this POU *)
    vTestCase1_act : WORD;  (* Test data 1 of test case 1 *)
    vTestCase1_xp : WORD;  (* Test data 2 of test case 1 *)
    vTestCase2_act : WORD;  (* Test data 1 of test case 2 *)
    vTestCase2_xp : WORD;  (* Test data 2 of test case 2 *)
  END_VAR

                    (*Run the test cases*)
TEST_CASE_1_SETUP();
TEST_CASE_1_EXEC();

TEST_CASE_2_SETUP();
TEST_CASE_2_EXEC();

(*Instantiate the test runner*)
testRunner(
	Id := 51,
	Name := 'assertGreater_WORD',
    RunTests := GVL.RunAll OR vRunAll,
	ResetTests := GVL.ResetAll OR vResetAll,
	TestCases:=vTestCases);

(*Report the results to the collection global*)
GVL.Results[testRunner.Id] := testRunner.Summary;
                  

ACTION TEST_CASE_2_SETUP:
                        IF vTestCases[1].state = utTestCaseStates.ut_SETUP THEN
	(*Setup the test case information*)
	vTestCases[1].id := 2;
    vTestCases[1].desc[0] := 'RETURNS FALSE WHEN PARAMETER ACT LESS THAN XP';
    vTestCases[1].desc[1] := 'Tests if the function returns False if the parameter act is less than parameter xp';
	vTestCases[1].desc[2] := 'PASS IF: Return value is FALSE';
	
	(*Setup needed variables*)
	vTestCase2_act := REAL_TO_WORD(8.4);
	vTestCase2_xp := REAL_TO_WORD(85.4);
END_IF
                      
END_ACTION

ACTION TEST_CASE_2_EXEC:
                        IF vTestCases[1].state = utTestCaseStates.ut_RUNNING THEN
	(*Run the test case*)
	IF NOT assertGreater_WORD(vTestCase2_act, vTestCase2_xp) THEN
		vTestCases[1].state := utTestCaseStates.ut_PASSED;
		vTestCases[1].msg := 'Parameter act was less than xp and function returned FALSE -> PASS';
	ELSE
		vTestCases[1].state := utTestCaseStates.ut_FAILED;
		vTestCases[1].msg := 'Parameter act was less than xp and function returned TRUE -> FAIL';
	END_IF
END_IF
                      
END_ACTION

ACTION TEST_CASE_1_SETUP:
                        IF vTestCases[0].state = utTestCaseStates.ut_SETUP THEN
	(*Setup the test case information*)
	vTestCases[0].id := 1;
	vTestCases[0].desc[0] := 'RETURNS TRUE WHEN PARAMETER ACT GREATER THAN XP';
    vTestCases[0].desc[1] := 'Tests if the function returns True if the parameter act is greater than parameter xp';
	vTestCases[0].desc[2] := 'PASS IF: Return value is TRUE';
	
	(*Setup needed variables*)
	vTestCase1_act := REAL_TO_WORD(115.4);
	vTestCase1_xp := REAL_TO_WORD(85.4);
END_IF
                      
END_ACTION

ACTION TEST_CASE_1_EXEC:
                        IF vTestCases[0].state = utTestCaseStates.ut_RUNNING THEN
	(*Run the test case*)
	IF assertGreater_WORD(vTestCase1_act, vTestCase1_xp) THEN
		vTestCases[0].state := utTestCaseStates.ut_PASSED;
		vTestCases[0].msg := 'Parameter act was greater than xp and function returned TRUE -> PASS';
	ELSE
		vTestCases[0].state := utTestCaseStates.ut_FAILED;
		vTestCases[0].msg := 'Parameter act was greater than xp and function returned FALSE -> FAIL';
	END_IF
END_IF
                      
END_ACTION
END_PROGRAM

PROGRAM test_assertNotEqual_TIME
  VAR
    vTestCases : ARRAY[0..20] OF utTestCase;  (* Definition of all test cases for this POU *)
    testRunner : utTestSuite;  (* Test Suite fb instance to run the tests *)
    vRunAll : BOOL;  (* Manual command to run all tests for this POU *)
    vResetAll : BOOL;  (* Manual command to reset all tests for this POU *)
    vTestCase1_act : TIME;  (* Test data 1 of test case 1 *)
    vTestCase1_xp : TIME;  (* Test data 2 of test case 1 *)
    vTestCase2_act : TIME;  (* Test data 1 of test case 2 *)
    vTestCase2_xp : TIME;  (* Test data 2 of test case 2 *)
  END_VAR

                    (*Run the test cases*)
TEST_CASE_1_SETUP();
TEST_CASE_1_EXEC();

TEST_CASE_2_SETUP();
TEST_CASE_2_EXEC();

(*Instantiate the test runner*)
testRunner(
	Id := 42,
	Name := 'assertNotEqual_TIME',
    RunTests := GVL.RunAll OR vRunAll,
	ResetTests := GVL.ResetAll OR vResetAll,
	TestCases:=vTestCases);

(*Report the results to the collection global*)
GVL.Results[testRunner.Id] := testRunner.Summary;
                  

ACTION TEST_CASE_1_SETUP:
                        IF vTestCases[0].state = utTestCaseStates.ut_SETUP THEN
	(*Setup the test case information*)
	vTestCases[0].id := 1;
	vTestCases[0].desc[0] := 'RETURNS TRUE WHEN PARAMETERS NOT EQUAL';
    vTestCases[0].desc[1] := 'Tests if the function returns True if the passed in parameters do not hold the same value';
	vTestCases[0].desc[2] := 'PASS IF: Return value is TRUE';
	
	(*Setup needed variables*)
	vTestCase1_act := REAL_TO_TIME(115.4);
	vTestCase1_xp := REAL_TO_TIME(-85.4);
END_IF
                      
END_ACTION

ACTION TEST_CASE_1_EXEC:
                        IF vTestCases[0].state = utTestCaseStates.ut_RUNNING THEN
	(*Run the test case*)
	IF assertNotEqual_TIME(vTestCase1_act, vTestCase1_xp) THEN
		vTestCases[0].state := utTestCaseStates.ut_PASSED;
		vTestCases[0].msg := 'Passed parameters were not equal and function returned TRUE -> PASS';
	ELSE
		vTestCases[0].state := utTestCaseStates.ut_FAILED;
		vTestCases[0].msg := 'Passed parameters were not equal and function returned FALSE -> FAIL';
	END_IF
END_IF
                      
END_ACTION

ACTION TEST_CASE_2_SETUP:
                        IF vTestCases[1].state = utTestCaseStates.ut_SETUP THEN
	(*Setup the test case information*)
	vTestCases[1].id := 2;
	vTestCases[1].desc[0] := 'RETURNS FALSE WHEN PARAMETERS EQUAL';
    vTestCases[1].desc[1] := 'Tests if the function returns False if the passed in parameters hold the same value';
	vTestCases[1].desc[2] := 'PASS IF: Return value is FALSE';
	
	(*Setup needed variables*)
	vTestCase2_act := REAL_TO_TIME(115.4);
	vTestCase2_xp := REAL_TO_TIME(115.4);
END_IF
                      
END_ACTION

ACTION TEST_CASE_2_EXEC:
                        IF vTestCases[1].state = utTestCaseStates.ut_RUNNING THEN
	(*Run the test case*)
	IF NOT assertNotEqual_TIME(vTestCase2_act, vTestCase2_xp) THEN
		vTestCases[1].state := utTestCaseStates.ut_PASSED;
		vTestCases[1].msg := 'Passed parameters were equal and function returned FALSE -> PASS';
	ELSE
		vTestCases[1].state := utTestCaseStates.ut_FAILED;
		vTestCases[1].msg := 'Passed parameters were equal and function returned TRUE -> FAIL';
	END_IF
END_IF
                      
END_ACTION
END_PROGRAM

PROGRAM test_assertNotEqual_LTIME
  VAR
    vTestCases : ARRAY[0..20] OF utTestCase;  (* Definition of all test cases for this POU *)
    testRunner : utTestSuite;  (* Test Suite fb instance to run the tests *)
    vRunAll : BOOL;  (* Manual command to run all tests for this POU *)
    vResetAll : BOOL;  (* Manual command to reset all tests for this POU *)
    vTestCase1_act : LTIME;  (* Test data 1 of test case 1 *)
    vTestCase1_xp : LTIME;  (* Test data 2 of test case 1 *)
    vTestCase2_act : LTIME;  (* Test data 1 of test case 2 *)
    vTestCase2_xp : LTIME;  (* Test data 2 of test case 2 *)
  END_VAR

                    (*Run the test cases*)
TEST_CASE_1_SETUP();
TEST_CASE_1_EXEC();

TEST_CASE_2_SETUP();
TEST_CASE_2_EXEC();

(*Instantiate the test runner*)
testRunner(
	Id := 43,
	Name := 'assertNotEqual_LTIME',
    RunTests := GVL.RunAll OR vRunAll,
	ResetTests := GVL.ResetAll OR vResetAll,
	TestCases:=vTestCases);

(*Report the results to the collection global*)
GVL.Results[testRunner.Id] := testRunner.Summary;
                  

ACTION TEST_CASE_1_SETUP:
                        IF vTestCases[0].state = utTestCaseStates.ut_SETUP THEN
	(*Setup the test case information*)
	vTestCases[0].id := 1;
	vTestCases[0].desc[0] := 'RETURNS TRUE WHEN PARAMETERS NOT EQUAL';
    vTestCases[0].desc[1] := 'Tests if the function returns True if the passed in parameters do not hold the same value';
	vTestCases[0].desc[2] := 'PASS IF: Return value is TRUE';
	
	(*Setup needed variables*)
	vTestCase1_act := REAL_TO_LTIME(115.4);
	vTestCase1_xp := REAL_TO_LTIME(-85.4);
END_IF
                      
END_ACTION

ACTION TEST_CASE_1_EXEC:
                        IF vTestCases[0].state = utTestCaseStates.ut_RUNNING THEN
	(*Run the test case*)
	IF assertNotEqual_LTIME(vTestCase1_act, vTestCase1_xp) THEN
		vTestCases[0].state := utTestCaseStates.ut_PASSED;
		vTestCases[0].msg := 'Passed parameters were not equal and function returned TRUE -> PASS';
	ELSE
		vTestCases[0].state := utTestCaseStates.ut_FAILED;
		vTestCases[0].msg := 'Passed parameters were not equal and function returned FALSE -> FAIL';
	END_IF
END_IF
                      
END_ACTION

ACTION TEST_CASE_2_SETUP:
                        IF vTestCases[1].state = utTestCaseStates.ut_SETUP THEN
	(*Setup the test case information*)
	vTestCases[1].id := 2;
	vTestCases[1].desc[0] := 'RETURNS FALSE WHEN PARAMETERS EQUAL';
    vTestCases[1].desc[1] := 'Tests if the function returns False if the passed in parameters hold the same value';
	vTestCases[1].desc[2] := 'PASS IF: Return value is FALSE';
	
	(*Setup needed variables*)
	vTestCase2_act := REAL_TO_LTIME(115.4);
	vTestCase2_xp := REAL_TO_LTIME(115.4);
END_IF
                      
END_ACTION

ACTION TEST_CASE_2_EXEC:
                        IF vTestCases[1].state = utTestCaseStates.ut_RUNNING THEN
	(*Run the test case*)
	IF NOT assertNotEqual_LTIME(vTestCase2_act, vTestCase2_xp) THEN
		vTestCases[1].state := utTestCaseStates.ut_PASSED;
		vTestCases[1].msg := 'Passed parameters were equal and function returned FALSE -> PASS';
	ELSE
		vTestCases[1].state := utTestCaseStates.ut_FAILED;
		vTestCases[1].msg := 'Passed parameters were equal and function returned TRUE -> FAIL';
	END_IF
END_IF
                      
END_ACTION
END_PROGRAM

PROGRAM test_assertGreaterEqual_LTIME_OF_DAY
  VAR
    vTestCases : ARRAY[0..20] OF utTestCase;  (* Definition of all test cases for this POU *)
    testRunner : utTestSuite;  (* Test Suite fb instance to run the tests *)
    vRunAll : BOOL;  (* Manual command to run all tests for this POU *)
    vResetAll : BOOL;  (* Manual command to reset all tests for this POU *)
    vTestCase1_act : LTIME_OF_DAY;  (* Test data 1 of test case 1 *)
    vTestCase1_xp : LTIME_OF_DAY;  (* Test data 2 of test case 1 *)
    vTestCase2_act : LTIME_OF_DAY;  (* Test data 1 of test case 2 *)
    vTestCase2_xp : LTIME_OF_DAY;  (* Test data 2 of test case 2 *)
    vTestCase3_act : LTIME_OF_DAY;  (* Test data 1 of test case 3 *)
    vTestCase3_xp : LTIME_OF_DAY;  (* Test data 2 of test case 3 *)
  END_VAR

                    (*Run the test cases*)
TEST_CASE_1_SETUP();
TEST_CASE_1_EXEC();

TEST_CASE_2_SETUP();
TEST_CASE_2_EXEC();

TEST_CASE_3_SETUP();
TEST_CASE_3_EXEC();

(*Instantiate the test runner*)
testRunner(
	Id := 93,
	Name := 'assertGreaterEqual_LTIME_OF_DAY',
    RunTests := GVL.RunAll OR vRunAll,
	ResetTests := GVL.ResetAll OR vResetAll,
	TestCases:=vTestCases);

(*Report the results to the collection global*)
GVL.Results[testRunner.Id] := testRunner.Summary;
                  

ACTION TEST_CASE_2_SETUP:
                        IF vTestCases[1].state = utTestCaseStates.ut_SETUP THEN
	(*Setup the test case information*)
	vTestCases[1].id := 2;
    vTestCases[1].desc[0] := 'RETURNS TRUE WHEN PARAMETER ACT EQUAL TO XP';
    vTestCases[1].desc[1] := 'Tests if the function returns True if the parameter act is equal to parameter xp';
	vTestCases[1].desc[2] := 'PASS IF: Return value is TRUE';
	
	(*Setup needed variables*)
	vTestCase2_act := REAL_TO_LTOD(115.4);
	vTestCase2_xp := REAL_TO_LTOD(115.4);
END_IF
                      
END_ACTION

ACTION TEST_CASE_3_SETUP:
                        IF vTestCases[2].state = utTestCaseStates.ut_SETUP THEN
	(*Setup the test case information*)
	vTestCases[2].id := 3;
    vTestCases[2].desc[0] := 'RETURNS FALSE WHEN PARAMETER ACT LESS THAN XP';
    vTestCases[2].desc[1] := 'Tests if the function returns False if the parameter act is less than parameter xp';
	vTestCases[2].desc[2] := 'PASS IF: Return value is FALSE';
	
	(*Setup needed variables*)
	vTestCase3_act := REAL_TO_LTOD(85.4);
	vTestCase3_xp := REAL_TO_LTOD(115.4);
END_IF
                      
END_ACTION

ACTION TEST_CASE_1_SETUP:
                        IF vTestCases[0].state = utTestCaseStates.ut_SETUP THEN
	(*Setup the test case information*)
	vTestCases[0].id := 1;
	vTestCases[0].desc[0] := 'RETURNS TRUE WHEN PARAMETER ACT GREATER THAN XP';
    vTestCases[0].desc[1] := 'Tests if the function returns True if the parameter act is greater than parameter xp';
	vTestCases[0].desc[2] := 'PASS IF: Return value is TRUE';
	
	(*Setup needed variables*)
	vTestCase1_act := REAL_TO_LTOD(115.4);
	vTestCase1_xp := REAL_TO_LTOD(85.4);
END_IF
                      
END_ACTION

ACTION TEST_CASE_1_EXEC:
                        IF vTestCases[0].state = utTestCaseStates.ut_RUNNING THEN
	(*Run the test case*)
	IF assertGreaterEqual_LTIME_OF_DAY(vTestCase1_act, vTestCase1_xp) THEN
		vTestCases[0].state := utTestCaseStates.ut_PASSED;
		vTestCases[0].msg := 'Parameter act was greater than xp and function returned TRUE -> PASS';
	ELSE
		vTestCases[0].state := utTestCaseStates.ut_FAILED;
		vTestCases[0].msg := 'Parameter act was greater than xp and function returned FALSE -> FAIL';
	END_IF
END_IF
                      
END_ACTION

ACTION TEST_CASE_2_EXEC:
                        IF vTestCases[1].state = utTestCaseStates.ut_RUNNING THEN
	(*Run the test case*)
	IF assertGreaterEqual_LTIME_OF_DAY(vTestCase2_act, vTestCase2_xp) THEN
		vTestCases[1].state := utTestCaseStates.ut_PASSED;
		vTestCases[1].msg := 'Parameter act was equal to xp and function returned TRUE -> PASS';
	ELSE
		vTestCases[1].state := utTestCaseStates.ut_FAILED;
		vTestCases[1].msg := 'Parameter act was equal to xp and function returned FALSE -> FAIL';
	END_IF
END_IF
                      
END_ACTION

ACTION TEST_CASE_3_EXEC:
                        IF vTestCases[2].state = utTestCaseStates.ut_RUNNING THEN
	(*Run the test case*)
	IF NOT assertGreaterEqual_LTIME_OF_DAY(vTestCase3_act, vTestCase3_xp) THEN
		vTestCases[2].state := utTestCaseStates.ut_PASSED;
		vTestCases[2].msg := 'Parameter act was less than xp and function returned FALSE -> PASS';
	ELSE
		vTestCases[2].state := utTestCaseStates.ut_FAILED;
		vTestCases[2].msg := 'Parameter act was less than xp and function returned TRUE -> FAIL';
	END_IF
END_IF
                      
END_ACTION
END_PROGRAM

PROGRAM test_assertLessEqual_INT
  VAR
    vTestCases : ARRAY[0..20] OF utTestCase;  (* Definition of all test cases for this POU *)
    testRunner : utTestSuite;  (* Test Suite fb instance to run the tests *)
    vRunAll : BOOL;  (* Manual command to run all tests for this POU *)
    vResetAll : BOOL;  (* Manual command to reset all tests for this POU *)
    vTestCase1_act : INT;  (* Test data 1 of test case 1 *)
    vTestCase1_xp : INT;  (* Test data 2 of test case 1 *)
    vTestCase2_act : INT;  (* Test data 1 of test case 2 *)
    vTestCase2_xp : INT;  (* Test data 2 of test case 2 *)
    vTestCase3_act : INT;  (* Test data 1 of test case 3 *)
    vTestCase3_xp : INT;  (* Test data 2 of test case 3 *)
  END_VAR

                    (*Run the test cases*)
TEST_CASE_1_SETUP();
TEST_CASE_1_EXEC();

TEST_CASE_2_SETUP();
TEST_CASE_2_EXEC();

TEST_CASE_3_SETUP();
TEST_CASE_3_EXEC();

(*Instantiate the test runner*)
testRunner(
	Id := 122,
	Name := 'assertLessEqual_INT',
    RunTests := GVL.RunAll OR vRunAll,
	ResetTests := GVL.ResetAll OR vResetAll,
	TestCases:=vTestCases);

(*Report the results to the collection global*)
GVL.Results[testRunner.Id] := testRunner.Summary;
                  

ACTION TEST_CASE_3_SETUP:
                        IF vTestCases[2].state = utTestCaseStates.ut_SETUP THEN
	(*Setup the test case information*)
	vTestCases[2].id := 3;
    vTestCases[2].desc[0] := 'RETURNS FALSE WHEN PARAMETER ACT GREATER THAN XP';
    vTestCases[2].desc[1] := 'Tests if the function returns False if the parameter act is greater than parameter xp';
	vTestCases[2].desc[2] := 'PASS IF: Return value is FALSE';
	
	(*Setup needed variables*)
	vTestCase3_act := REAL_TO_INT(115.4);
	vTestCase3_xp := REAL_TO_INT(85.4);
END_IF
                      
END_ACTION

ACTION TEST_CASE_1_SETUP:
                        IF vTestCases[0].state = utTestCaseStates.ut_SETUP THEN
	(*Setup the test case information*)
	vTestCases[0].id := 1;
	vTestCases[0].desc[0] := 'RETURNS TRUE WHEN PARAMETER ACT LESS THAN XP';
    vTestCases[0].desc[1] := 'Tests if the function returns True if the parameter act is less than parameter xp';
	vTestCases[0].desc[2] := 'PASS IF: Return value is TRUE';
	
	(*Setup needed variables*)
	vTestCase1_act := REAL_TO_INT(85.4);
	vTestCase1_xp := REAL_TO_INT(115.4);
END_IF
                      
END_ACTION

ACTION TEST_CASE_1_EXEC:
                        IF vTestCases[0].state = utTestCaseStates.ut_RUNNING THEN
	(*Run the test case*)
	IF assertLessEqual_INT(vTestCase1_act, vTestCase1_xp) THEN
		vTestCases[0].state := utTestCaseStates.ut_PASSED;
		vTestCases[0].msg := 'Parameter act was less than xp and function returned TRUE -> PASS';
	ELSE
		vTestCases[0].state := utTestCaseStates.ut_FAILED;
		vTestCases[0].msg := 'Parameter act was less than xp and function returned FALSE -> FAIL';
	END_IF
END_IF
                      
END_ACTION

ACTION TEST_CASE_2_SETUP:
                        IF vTestCases[1].state = utTestCaseStates.ut_SETUP THEN
	(*Setup the test case information*)
	vTestCases[1].id := 2;
    vTestCases[1].desc[0] := 'RETURNS TRUE WHEN PARAMETER ACT EQUAL TO XP';
    vTestCases[1].desc[1] := 'Tests if the function returns True if the parameter act is equal to parameter xp';
	vTestCases[1].desc[2] := 'PASS IF: Return value is TRUE';
	
	(*Setup needed variables*)
	vTestCase2_act := REAL_TO_INT(115.4);
	vTestCase2_xp := REAL_TO_INT(115.4);
END_IF
                      
END_ACTION

ACTION TEST_CASE_2_EXEC:
                        IF vTestCases[1].state = utTestCaseStates.ut_RUNNING THEN
	(*Run the test case*)
	IF assertLessEqual_INT(vTestCase2_act, vTestCase2_xp) THEN
		vTestCases[1].state := utTestCaseStates.ut_PASSED;
		vTestCases[1].msg := 'Parameter act was equal to xp and function returned TRUE -> PASS';
	ELSE
		vTestCases[1].state := utTestCaseStates.ut_FAILED;
		vTestCases[1].msg := 'Parameter act was equal to xp and function returned FALSE -> FAIL';
	END_IF
END_IF
                      
END_ACTION

ACTION TEST_CASE_3_EXEC:
                        IF vTestCases[2].state = utTestCaseStates.ut_RUNNING THEN
	(*Run the test case*)
	IF NOT assertLessEqual_INT(vTestCase3_act, vTestCase3_xp) THEN
		vTestCases[2].state := utTestCaseStates.ut_PASSED;
		vTestCases[2].msg := 'Parameter act was greater than xp and function returned FALSE -> PASS';
	ELSE
		vTestCases[2].state := utTestCaseStates.ut_FAILED;
		vTestCases[2].msg := 'Parameter act was greater than xp and function returned TRUE -> FAIL';
	END_IF
END_IF
                      
END_ACTION
END_PROGRAM

PROGRAM test_assertLess_SINT
  VAR
    vTestCases : ARRAY[0..20] OF utTestCase;  (* Definition of all test cases for this POU *)
    testRunner : utTestSuite;  (* Test Suite fb instance to run the tests *)
    vRunAll : BOOL;  (* Manual command to run all tests for this POU *)
    vResetAll : BOOL;  (* Manual command to reset all tests for this POU *)
    vTestCase1_act : SINT;  (* Test data 1 of test case 1 *)
    vTestCase1_xp : SINT;  (* Test data 2 of test case 1 *)
    vTestCase2_act : SINT;  (* Test data 1 of test case 2 *)
    vTestCase2_xp : SINT;  (* Test data 2 of test case 2 *)
  END_VAR

                    (*Run the test cases*)
TEST_CASE_1_SETUP();
TEST_CASE_1_EXEC();

TEST_CASE_2_SETUP();
TEST_CASE_2_EXEC();

(*Instantiate the test runner*)
testRunner(
	Id := 98,
	Name := 'assertLess_SINT',
    RunTests := GVL.RunAll OR vRunAll,
	ResetTests := GVL.ResetAll OR vResetAll,
	TestCases:=vTestCases);

(*Report the results to the collection global*)
GVL.Results[testRunner.Id] := testRunner.Summary;
                  

ACTION TEST_CASE_1_SETUP:
                        IF vTestCases[0].state = utTestCaseStates.ut_SETUP THEN
	(*Setup the test case information*)
	vTestCases[0].id := 1;
	vTestCases[0].desc[0] := 'RETURNS TRUE WHEN PARAMETER ACT LESS THAN XP';
    vTestCases[0].desc[1] := 'Tests if the function returns True if the parameter act is less than parameter xp';
	vTestCases[0].desc[2] := 'PASS IF: Return value is TRUE';
	
	(*Setup needed variables*)
	vTestCase1_act := REAL_TO_SINT(85.4);
	vTestCase1_xp := REAL_TO_SINT(115.4);
END_IF
                      
END_ACTION

ACTION TEST_CASE_1_EXEC:
                        IF vTestCases[0].state = utTestCaseStates.ut_RUNNING THEN
	(*Run the test case*)
	IF assertLess_SINT(vTestCase1_act, vTestCase1_xp) THEN
		vTestCases[0].state := utTestCaseStates.ut_PASSED;
		vTestCases[0].msg := 'Parameter act was less than xp and function returned TRUE -> PASS';
	ELSE
		vTestCases[0].state := utTestCaseStates.ut_FAILED;
		vTestCases[0].msg := 'Parameter act was less than xp and function returned FALSE -> FAIL';
	END_IF
END_IF
                      
END_ACTION

ACTION TEST_CASE_2_SETUP:
                        IF vTestCases[1].state = utTestCaseStates.ut_SETUP THEN
	(*Setup the test case information*)
	vTestCases[1].id := 2;
    vTestCases[1].desc[0] := 'RETURNS FALSE WHEN PARAMETER ACT GREATER THAN XP';
    vTestCases[1].desc[1] := 'Tests if the function returns False if the parameter act is greater than parameter xp';
	vTestCases[1].desc[2] := 'PASS IF: Return value is FALSE';
	
	(*Setup needed variables*)
	vTestCase2_act := REAL_TO_SINT(115.4);
	vTestCase2_xp := REAL_TO_SINT(85.4);
END_IF
                      
END_ACTION

ACTION TEST_CASE_2_EXEC:
                        IF vTestCases[1].state = utTestCaseStates.ut_RUNNING THEN
	(*Run the test case*)
	IF NOT assertLess_SINT(vTestCase2_act, vTestCase2_xp) THEN
		vTestCases[1].state := utTestCaseStates.ut_PASSED;
		vTestCases[1].msg := 'Parameter act was greater than xp and function returned FALSE -> PASS';
	ELSE
		vTestCases[1].state := utTestCaseStates.ut_FAILED;
		vTestCases[1].msg := 'Parameter act was greater than xp and function returned TRUE -> FAIL';
	END_IF
END_IF
                      
END_ACTION
END_PROGRAM

PROGRAM test_assertLess_USINT
  VAR
    vTestCases : ARRAY[0..20] OF utTestCase;  (* Definition of all test cases for this POU *)
    testRunner : utTestSuite;  (* Test Suite fb instance to run the tests *)
    vRunAll : BOOL;  (* Manual command to run all tests for this POU *)
    vResetAll : BOOL;  (* Manual command to reset all tests for this POU *)
    vTestCase1_act : USINT;  (* Test data 1 of test case 1 *)
    vTestCase1_xp : USINT;  (* Test data 2 of test case 1 *)
    vTestCase2_act : USINT;  (* Test data 1 of test case 2 *)
    vTestCase2_xp : USINT;  (* Test data 2 of test case 2 *)
  END_VAR

                    (*Run the test cases*)
TEST_CASE_1_SETUP();
TEST_CASE_1_EXEC();

TEST_CASE_2_SETUP();
TEST_CASE_2_EXEC();

(*Instantiate the test runner*)
testRunner(
	Id := 99,
	Name := 'assertLess_USINT',
    RunTests := GVL.RunAll OR vRunAll,
	ResetTests := GVL.ResetAll OR vResetAll,
	TestCases:=vTestCases);

(*Report the results to the collection global*)
GVL.Results[testRunner.Id] := testRunner.Summary;
                  

ACTION TEST_CASE_1_SETUP:
                        IF vTestCases[0].state = utTestCaseStates.ut_SETUP THEN
	(*Setup the test case information*)
	vTestCases[0].id := 1;
	vTestCases[0].desc[0] := 'RETURNS TRUE WHEN PARAMETER ACT LESS THAN XP';
    vTestCases[0].desc[1] := 'Tests if the function returns True if the parameter act is less than parameter xp';
	vTestCases[0].desc[2] := 'PASS IF: Return value is TRUE';
	
	(*Setup needed variables*)
	vTestCase1_act := REAL_TO_USINT(85.4);
	vTestCase1_xp := REAL_TO_USINT(115.4);
END_IF
                      
END_ACTION

ACTION TEST_CASE_1_EXEC:
                        IF vTestCases[0].state = utTestCaseStates.ut_RUNNING THEN
	(*Run the test case*)
	IF assertLess_USINT(vTestCase1_act, vTestCase1_xp) THEN
		vTestCases[0].state := utTestCaseStates.ut_PASSED;
		vTestCases[0].msg := 'Parameter act was less than xp and function returned TRUE -> PASS';
	ELSE
		vTestCases[0].state := utTestCaseStates.ut_FAILED;
		vTestCases[0].msg := 'Parameter act was less than xp and function returned FALSE -> FAIL';
	END_IF
END_IF
                      
END_ACTION

ACTION TEST_CASE_2_SETUP:
                        IF vTestCases[1].state = utTestCaseStates.ut_SETUP THEN
	(*Setup the test case information*)
	vTestCases[1].id := 2;
    vTestCases[1].desc[0] := 'RETURNS FALSE WHEN PARAMETER ACT GREATER THAN XP';
    vTestCases[1].desc[1] := 'Tests if the function returns False if the parameter act is greater than parameter xp';
	vTestCases[1].desc[2] := 'PASS IF: Return value is FALSE';
	
	(*Setup needed variables*)
	vTestCase2_act := REAL_TO_USINT(115.4);
	vTestCase2_xp := REAL_TO_USINT(85.4);
END_IF
                      
END_ACTION

ACTION TEST_CASE_2_EXEC:
                        IF vTestCases[1].state = utTestCaseStates.ut_RUNNING THEN
	(*Run the test case*)
	IF NOT assertLess_USINT(vTestCase2_act, vTestCase2_xp) THEN
		vTestCases[1].state := utTestCaseStates.ut_PASSED;
		vTestCases[1].msg := 'Parameter act was greater than xp and function returned FALSE -> PASS';
	ELSE
		vTestCases[1].state := utTestCaseStates.ut_FAILED;
		vTestCases[1].msg := 'Parameter act was greater than xp and function returned TRUE -> FAIL';
	END_IF
END_IF
                      
END_ACTION
END_PROGRAM

PROGRAM test_assertLess_DATE
  VAR
    vTestCases : ARRAY[0..20] OF utTestCase;  (* Definition of all test cases for this POU *)
    testRunner : utTestSuite;  (* Test Suite fb instance to run the tests *)
    vRunAll : BOOL;  (* Manual command to run all tests for this POU *)
    vResetAll : BOOL;  (* Manual command to reset all tests for this POU *)
    vTestCase1_act : DATE;  (* Test data 1 of test case 1 *)
    vTestCase1_xp : DATE;  (* Test data 2 of test case 1 *)
    vTestCase2_act : DATE;  (* Test data 1 of test case 2 *)
    vTestCase2_xp : DATE;  (* Test data 2 of test case 2 *)
  END_VAR

                    (*Run the test cases*)
TEST_CASE_1_SETUP();
TEST_CASE_1_EXEC();

TEST_CASE_2_SETUP();
TEST_CASE_2_EXEC();

(*Instantiate the test runner*)
testRunner(
	Id := 110,
	Name := 'assertLess_DATE',
    RunTests := GVL.RunAll OR vRunAll,
	ResetTests := GVL.ResetAll OR vResetAll,
	TestCases:=vTestCases);

(*Report the results to the collection global*)
GVL.Results[testRunner.Id] := testRunner.Summary;
                  

ACTION TEST_CASE_1_EXEC:
                        IF vTestCases[0].state = utTestCaseStates.ut_RUNNING THEN
	(*Run the test case*)
	IF assertLess_DATE(vTestCase1_act, vTestCase1_xp) THEN
		vTestCases[0].state := utTestCaseStates.ut_PASSED;
		vTestCases[0].msg := 'Parameter act was less than xp and function returned TRUE -> PASS';
	ELSE
		vTestCases[0].state := utTestCaseStates.ut_FAILED;
		vTestCases[0].msg := 'Parameter act was less than xp and function returned FALSE -> FAIL';
	END_IF
END_IF
                      
END_ACTION

ACTION TEST_CASE_1_SETUP:
                        IF vTestCases[0].state = utTestCaseStates.ut_SETUP THEN
	(*Setup the test case information*)
	vTestCases[0].id := 1;
	vTestCases[0].desc[0] := 'RETURNS TRUE WHEN PARAMETER ACT LESS THAN XP';
    vTestCases[0].desc[1] := 'Tests if the function returns True if the parameter act is less than parameter xp';
	vTestCases[0].desc[2] := 'PASS IF: Return value is TRUE';
	
	(*Setup needed variables*)
	vTestCase1_act := REAL_TO_DATE(85.4);
	vTestCase1_xp := REAL_TO_DATE(115.4);
END_IF
                      
END_ACTION

ACTION TEST_CASE_2_SETUP:
                        IF vTestCases[1].state = utTestCaseStates.ut_SETUP THEN
	(*Setup the test case information*)
	vTestCases[1].id := 2;
    vTestCases[1].desc[0] := 'RETURNS FALSE WHEN PARAMETER ACT GREATER THAN XP';
    vTestCases[1].desc[1] := 'Tests if the function returns False if the parameter act is greater than parameter xp';
	vTestCases[1].desc[2] := 'PASS IF: Return value is FALSE';
	
	(*Setup needed variables*)
	vTestCase2_act := REAL_TO_DATE(115.4);
	vTestCase2_xp := REAL_TO_DATE(85.4);
END_IF
                      
END_ACTION

ACTION TEST_CASE_2_EXEC:
                        IF vTestCases[1].state = utTestCaseStates.ut_RUNNING THEN
	(*Run the test case*)
	IF NOT assertLess_DATE(vTestCase2_act, vTestCase2_xp) THEN
		vTestCases[1].state := utTestCaseStates.ut_PASSED;
		vTestCases[1].msg := 'Parameter act was greater than xp and function returned FALSE -> PASS';
	ELSE
		vTestCases[1].state := utTestCaseStates.ut_FAILED;
		vTestCases[1].msg := 'Parameter act was greater than xp and function returned TRUE -> FAIL';
	END_IF
END_IF
                      
END_ACTION
END_PROGRAM

PROGRAM test_assertLess_DATE_AND_TIME
  VAR
    vTestCases : ARRAY[0..20] OF utTestCase;  (* Definition of all test cases for this POU *)
    testRunner : utTestSuite;  (* Test Suite fb instance to run the tests *)
    vRunAll : BOOL;  (* Manual command to run all tests for this POU *)
    vResetAll : BOOL;  (* Manual command to reset all tests for this POU *)
    vTestCase1_act : DT;  (* Test data 1 of test case 1 *)
    vTestCase1_xp : DT;  (* Test data 2 of test case 1 *)
    vTestCase2_act : DT;  (* Test data 1 of test case 2 *)
    vTestCase2_xp : DT;  (* Test data 2 of test case 2 *)
  END_VAR

                    (*Run the test cases*)
TEST_CASE_1_SETUP();
TEST_CASE_1_EXEC();

TEST_CASE_2_SETUP();
TEST_CASE_2_EXEC();

(*Instantiate the test runner*)
testRunner(
	Id := 112,
	Name := 'assertLess_DATE_AND_TIME',
    RunTests := GVL.RunAll OR vRunAll,
	ResetTests := GVL.ResetAll OR vResetAll,
	TestCases:=vTestCases);

(*Report the results to the collection global*)
GVL.Results[testRunner.Id] := testRunner.Summary;
                  

ACTION TEST_CASE_1_SETUP:
                        IF vTestCases[0].state = utTestCaseStates.ut_SETUP THEN
	(*Setup the test case information*)
	vTestCases[0].id := 1;
	vTestCases[0].desc[0] := 'RETURNS TRUE WHEN PARAMETER ACT LESS THAN XP';
    vTestCases[0].desc[1] := 'Tests if the function returns True if the parameter act is less than parameter xp';
	vTestCases[0].desc[2] := 'PASS IF: Return value is TRUE';
	
	(*Setup needed variables*)
	vTestCase1_act := REAL_TO_DT(85.4);
	vTestCase1_xp := REAL_TO_DT(115.4);
END_IF
                      
END_ACTION

ACTION TEST_CASE_1_EXEC:
                        IF vTestCases[0].state = utTestCaseStates.ut_RUNNING THEN
	(*Run the test case*)
	IF assertLess_DATE_AND_TIME(vTestCase1_act, vTestCase1_xp) THEN
		vTestCases[0].state := utTestCaseStates.ut_PASSED;
		vTestCases[0].msg := 'Parameter act was less than xp and function returned TRUE -> PASS';
	ELSE
		vTestCases[0].state := utTestCaseStates.ut_FAILED;
		vTestCases[0].msg := 'Parameter act was less than xp and function returned FALSE -> FAIL';
	END_IF
END_IF
                      
END_ACTION

ACTION TEST_CASE_2_SETUP:
                        IF vTestCases[1].state = utTestCaseStates.ut_SETUP THEN
	(*Setup the test case information*)
	vTestCases[1].id := 2;
    vTestCases[1].desc[0] := 'RETURNS FALSE WHEN PARAMETER ACT GREATER THAN XP';
    vTestCases[1].desc[1] := 'Tests if the function returns False if the parameter act is greater than parameter xp';
	vTestCases[1].desc[2] := 'PASS IF: Return value is FALSE';
	
	(*Setup needed variables*)
	vTestCase2_act := REAL_TO_DT(115.4);
	vTestCase2_xp := REAL_TO_DT(85.4);
END_IF
                      
END_ACTION

ACTION TEST_CASE_2_EXEC:
                        IF vTestCases[1].state = utTestCaseStates.ut_RUNNING THEN
	(*Run the test case*)
	IF NOT assertLess_DATE_AND_TIME(vTestCase2_act, vTestCase2_xp) THEN
		vTestCases[1].state := utTestCaseStates.ut_PASSED;
		vTestCases[1].msg := 'Parameter act was greater than xp and function returned FALSE -> PASS';
	ELSE
		vTestCases[1].state := utTestCaseStates.ut_FAILED;
		vTestCases[1].msg := 'Parameter act was greater than xp and function returned TRUE -> FAIL';
	END_IF
END_IF
                      
END_ACTION
END_PROGRAM

PROGRAM test_assertLess_LDATE_AND_TIME
  VAR
    vTestCases : ARRAY[0..20] OF utTestCase;  (* Definition of all test cases for this POU *)
    testRunner : utTestSuite;  (* Test Suite fb instance to run the tests *)
    vRunAll : BOOL;  (* Manual command to run all tests for this POU *)
    vResetAll : BOOL;  (* Manual command to reset all tests for this POU *)
    vTestCase1_act : LDATE_AND_TIME;  (* Test data 1 of test case 1 *)
    vTestCase1_xp : LDATE_AND_TIME;  (* Test data 2 of test case 1 *)
    vTestCase2_act : LDATE_AND_TIME;  (* Test data 1 of test case 2 *)
    vTestCase2_xp : LDATE_AND_TIME;  (* Test data 2 of test case 2 *)
  END_VAR

                    (*Run the test cases*)
TEST_CASE_1_SETUP();
TEST_CASE_1_EXEC();

TEST_CASE_2_SETUP();
TEST_CASE_2_EXEC();

(*Instantiate the test runner*)
testRunner(
	Id := 113,
	Name := 'assertLess_LDATE_AND_TIME',
    RunTests := GVL.RunAll OR vRunAll,
	ResetTests := GVL.ResetAll OR vResetAll,
	TestCases:=vTestCases);

(*Report the results to the collection global*)
GVL.Results[testRunner.Id] := testRunner.Summary;
                  

ACTION TEST_CASE_1_SETUP:
                        IF vTestCases[0].state = utTestCaseStates.ut_SETUP THEN
	(*Setup the test case information*)
	vTestCases[0].id := 1;
	vTestCases[0].desc[0] := 'RETURNS TRUE WHEN PARAMETER ACT LESS THAN XP';
    vTestCases[0].desc[1] := 'Tests if the function returns True if the parameter act is less than parameter xp';
	vTestCases[0].desc[2] := 'PASS IF: Return value is TRUE';
	
	(*Setup needed variables*)
	vTestCase1_act := REAL_TO_LDT(85.4);
	vTestCase1_xp := REAL_TO_LDT(115.4);
END_IF
                      
END_ACTION

ACTION TEST_CASE_1_EXEC:
                        IF vTestCases[0].state = utTestCaseStates.ut_RUNNING THEN
	(*Run the test case*)
	IF assertLess_LDATE_AND_TIME(vTestCase1_act, vTestCase1_xp) THEN
		vTestCases[0].state := utTestCaseStates.ut_PASSED;
		vTestCases[0].msg := 'Parameter act was less than xp and function returned TRUE -> PASS';
	ELSE
		vTestCases[0].state := utTestCaseStates.ut_FAILED;
		vTestCases[0].msg := 'Parameter act was less than xp and function returned FALSE -> FAIL';
	END_IF
END_IF
                      
END_ACTION

ACTION TEST_CASE_2_SETUP:
                        IF vTestCases[1].state = utTestCaseStates.ut_SETUP THEN
	(*Setup the test case information*)
	vTestCases[1].id := 2;
    vTestCases[1].desc[0] := 'RETURNS FALSE WHEN PARAMETER ACT GREATER THAN XP';
    vTestCases[1].desc[1] := 'Tests if the function returns False if the parameter act is greater than parameter xp';
	vTestCases[1].desc[2] := 'PASS IF: Return value is FALSE';
	
	(*Setup needed variables*)
	vTestCase2_act := REAL_TO_LDT(115.4);
	vTestCase2_xp := REAL_TO_LDT(85.4);
END_IF
                      
END_ACTION

ACTION TEST_CASE_2_EXEC:
                        IF vTestCases[1].state = utTestCaseStates.ut_RUNNING THEN
	(*Run the test case*)
	IF NOT assertLess_LDATE_AND_TIME(vTestCase2_act, vTestCase2_xp) THEN
		vTestCases[1].state := utTestCaseStates.ut_PASSED;
		vTestCases[1].msg := 'Parameter act was greater than xp and function returned FALSE -> PASS';
	ELSE
		vTestCases[1].state := utTestCaseStates.ut_FAILED;
		vTestCases[1].msg := 'Parameter act was greater than xp and function returned TRUE -> FAIL';
	END_IF
END_IF
                      
END_ACTION
END_PROGRAM

PROGRAM test_assertLessEqual_USINT
  VAR
    vTestCases : ARRAY[0..20] OF utTestCase;  (* Definition of all test cases for this POU *)
    testRunner : utTestSuite;  (* Test Suite fb instance to run the tests *)
    vRunAll : BOOL;  (* Manual command to run all tests for this POU *)
    vResetAll : BOOL;  (* Manual command to reset all tests for this POU *)
    vTestCase1_act : USINT;  (* Test data 1 of test case 1 *)
    vTestCase1_xp : USINT;  (* Test data 2 of test case 1 *)
    vTestCase2_act : USINT;  (* Test data 1 of test case 2 *)
    vTestCase2_xp : USINT;  (* Test data 2 of test case 2 *)
    vTestCase3_act : USINT;  (* Test data 1 of test case 3 *)
    vTestCase3_xp : USINT;  (* Test data 2 of test case 3 *)
  END_VAR

                    (*Run the test cases*)
TEST_CASE_1_SETUP();
TEST_CASE_1_EXEC();

TEST_CASE_2_SETUP();
TEST_CASE_2_EXEC();

TEST_CASE_3_SETUP();
TEST_CASE_3_EXEC();

(*Instantiate the test runner*)
testRunner(
	Id := 121,
	Name := 'assertLessEqual_USINT',
    RunTests := GVL.RunAll OR vRunAll,
	ResetTests := GVL.ResetAll OR vResetAll,
	TestCases:=vTestCases);

(*Report the results to the collection global*)
GVL.Results[testRunner.Id] := testRunner.Summary;
                  

ACTION TEST_CASE_2_SETUP:
                        IF vTestCases[1].state = utTestCaseStates.ut_SETUP THEN
	(*Setup the test case information*)
	vTestCases[1].id := 2;
    vTestCases[1].desc[0] := 'RETURNS TRUE WHEN PARAMETER ACT EQUAL TO XP';
    vTestCases[1].desc[1] := 'Tests if the function returns True if the parameter act is equal to parameter xp';
	vTestCases[1].desc[2] := 'PASS IF: Return value is TRUE';
	
	(*Setup needed variables*)
	vTestCase2_act := REAL_TO_USINT(115.4);
	vTestCase2_xp := REAL_TO_USINT(115.4);
END_IF
                      
END_ACTION

ACTION TEST_CASE_2_EXEC:
                        IF vTestCases[1].state = utTestCaseStates.ut_RUNNING THEN
	(*Run the test case*)
	IF assertLessEqual_USINT(vTestCase2_act, vTestCase2_xp) THEN
		vTestCases[1].state := utTestCaseStates.ut_PASSED;
		vTestCases[1].msg := 'Parameter act was equal to xp and function returned TRUE -> PASS';
	ELSE
		vTestCases[1].state := utTestCaseStates.ut_FAILED;
		vTestCases[1].msg := 'Parameter act was equal to xp and function returned FALSE -> FAIL';
	END_IF
END_IF
                      
END_ACTION

ACTION TEST_CASE_1_SETUP:
                        IF vTestCases[0].state = utTestCaseStates.ut_SETUP THEN
	(*Setup the test case information*)
	vTestCases[0].id := 1;
	vTestCases[0].desc[0] := 'RETURNS TRUE WHEN PARAMETER ACT LESS THAN XP';
    vTestCases[0].desc[1] := 'Tests if the function returns True if the parameter act is less than parameter xp';
	vTestCases[0].desc[2] := 'PASS IF: Return value is TRUE';
	
	(*Setup needed variables*)
	vTestCase1_act := REAL_TO_USINT(85.4);
	vTestCase1_xp := REAL_TO_USINT(115.4);
END_IF
                      
END_ACTION

ACTION TEST_CASE_1_EXEC:
                        IF vTestCases[0].state = utTestCaseStates.ut_RUNNING THEN
	(*Run the test case*)
	IF assertLessEqual_USINT(vTestCase1_act, vTestCase1_xp) THEN
		vTestCases[0].state := utTestCaseStates.ut_PASSED;
		vTestCases[0].msg := 'Parameter act was less than xp and function returned TRUE -> PASS';
	ELSE
		vTestCases[0].state := utTestCaseStates.ut_FAILED;
		vTestCases[0].msg := 'Parameter act was less than xp and function returned FALSE -> FAIL';
	END_IF
END_IF
                      
END_ACTION

ACTION TEST_CASE_3_SETUP:
                        IF vTestCases[2].state = utTestCaseStates.ut_SETUP THEN
	(*Setup the test case information*)
	vTestCases[2].id := 3;
    vTestCases[2].desc[0] := 'RETURNS FALSE WHEN PARAMETER ACT GREATER THAN XP';
    vTestCases[2].desc[1] := 'Tests if the function returns False if the parameter act is greater than parameter xp';
	vTestCases[2].desc[2] := 'PASS IF: Return value is FALSE';
	
	(*Setup needed variables*)
	vTestCase3_act := REAL_TO_USINT(115.4);
	vTestCase3_xp := REAL_TO_USINT(85.4);
END_IF
                      
END_ACTION

ACTION TEST_CASE_3_EXEC:
                        IF vTestCases[2].state = utTestCaseStates.ut_RUNNING THEN
	(*Run the test case*)
	IF NOT assertLessEqual_USINT(vTestCase3_act, vTestCase3_xp) THEN
		vTestCases[2].state := utTestCaseStates.ut_PASSED;
		vTestCases[2].msg := 'Parameter act was greater than xp and function returned FALSE -> PASS';
	ELSE
		vTestCases[2].state := utTestCaseStates.ut_FAILED;
		vTestCases[2].msg := 'Parameter act was greater than xp and function returned TRUE -> FAIL';
	END_IF
END_IF
                      
END_ACTION
END_PROGRAM

PROGRAM test_assertLess_INT
  VAR
    vTestCases : ARRAY[0..20] OF utTestCase;  (* Definition of all test cases for this POU *)
    testRunner : utTestSuite;  (* Test Suite fb instance to run the tests *)
    vRunAll : BOOL;  (* Manual command to run all tests for this POU *)
    vResetAll : BOOL;  (* Manual command to reset all tests for this POU *)
    vTestCase1_act : INT;  (* Test data 1 of test case 1 *)
    vTestCase1_xp : INT;  (* Test data 2 of test case 1 *)
    vTestCase2_act : INT;  (* Test data 1 of test case 2 *)
    vTestCase2_xp : INT;  (* Test data 2 of test case 2 *)
  END_VAR

                    (*Run the test cases*)
TEST_CASE_1_SETUP();
TEST_CASE_1_EXEC();

TEST_CASE_2_SETUP();
TEST_CASE_2_EXEC();

(*Instantiate the test runner*)
testRunner(
	Id := 100,
	Name := 'assertLess_INT',
    RunTests := GVL.RunAll OR vRunAll,
	ResetTests := GVL.ResetAll OR vResetAll,
	TestCases:=vTestCases);

(*Report the results to the collection global*)
GVL.Results[testRunner.Id] := testRunner.Summary;
                  

ACTION TEST_CASE_2_SETUP:
                        IF vTestCases[1].state = utTestCaseStates.ut_SETUP THEN
	(*Setup the test case information*)
	vTestCases[1].id := 2;
    vTestCases[1].desc[0] := 'RETURNS FALSE WHEN PARAMETER ACT GREATER THAN XP';
    vTestCases[1].desc[1] := 'Tests if the function returns False if the parameter act is greater than parameter xp';
	vTestCases[1].desc[2] := 'PASS IF: Return value is FALSE';
	
	(*Setup needed variables*)
	vTestCase2_act := REAL_TO_INT(115.4);
	vTestCase2_xp := REAL_TO_INT(85.4);
END_IF
                      
END_ACTION

ACTION TEST_CASE_1_SETUP:
                        IF vTestCases[0].state = utTestCaseStates.ut_SETUP THEN
	(*Setup the test case information*)
	vTestCases[0].id := 1;
	vTestCases[0].desc[0] := 'RETURNS TRUE WHEN PARAMETER ACT LESS THAN XP';
    vTestCases[0].desc[1] := 'Tests if the function returns True if the parameter act is less than parameter xp';
	vTestCases[0].desc[2] := 'PASS IF: Return value is TRUE';
	
	(*Setup needed variables*)
	vTestCase1_act := REAL_TO_INT(85.4);
	vTestCase1_xp := REAL_TO_INT(115.4);
END_IF
                      
END_ACTION

ACTION TEST_CASE_1_EXEC:
                        IF vTestCases[0].state = utTestCaseStates.ut_RUNNING THEN
	(*Run the test case*)
	IF assertLess_INT(vTestCase1_act, vTestCase1_xp) THEN
		vTestCases[0].state := utTestCaseStates.ut_PASSED;
		vTestCases[0].msg := 'Parameter act was less than xp and function returned TRUE -> PASS';
	ELSE
		vTestCases[0].state := utTestCaseStates.ut_FAILED;
		vTestCases[0].msg := 'Parameter act was less than xp and function returned FALSE -> FAIL';
	END_IF
END_IF
                      
END_ACTION

ACTION TEST_CASE_2_EXEC:
                        IF vTestCases[1].state = utTestCaseStates.ut_RUNNING THEN
	(*Run the test case*)
	IF NOT assertLess_INT(vTestCase2_act, vTestCase2_xp) THEN
		vTestCases[1].state := utTestCaseStates.ut_PASSED;
		vTestCases[1].msg := 'Parameter act was greater than xp and function returned FALSE -> PASS';
	ELSE
		vTestCases[1].state := utTestCaseStates.ut_FAILED;
		vTestCases[1].msg := 'Parameter act was greater than xp and function returned TRUE -> FAIL';
	END_IF
END_IF
                      
END_ACTION
END_PROGRAM

PROGRAM test_assertLessEqual_DWORD
  VAR
    vTestCases : ARRAY[0..20] OF utTestCase;  (* Definition of all test cases for this POU *)
    testRunner : utTestSuite;  (* Test Suite fb instance to run the tests *)
    vRunAll : BOOL;  (* Manual command to run all tests for this POU *)
    vResetAll : BOOL;  (* Manual command to reset all tests for this POU *)
    vTestCase1_act : DWORD;  (* Test data 1 of test case 1 *)
    vTestCase1_xp : DWORD;  (* Test data 2 of test case 1 *)
    vTestCase2_act : DWORD;  (* Test data 1 of test case 2 *)
    vTestCase2_xp : DWORD;  (* Test data 2 of test case 2 *)
    vTestCase3_act : DWORD;  (* Test data 1 of test case 3 *)
    vTestCase3_xp : DWORD;  (* Test data 2 of test case 3 *)
  END_VAR

                    (*Run the test cases*)
TEST_CASE_1_SETUP();
TEST_CASE_1_EXEC();

TEST_CASE_2_SETUP();
TEST_CASE_2_EXEC();

TEST_CASE_3_SETUP();
TEST_CASE_3_EXEC();

(*Instantiate the test runner*)
testRunner(
	Id := 118,
	Name := 'assertLessEqual_DWORD',
    RunTests := GVL.RunAll OR vRunAll,
	ResetTests := GVL.ResetAll OR vResetAll,
	TestCases:=vTestCases);

(*Report the results to the collection global*)
GVL.Results[testRunner.Id] := testRunner.Summary;
                  

ACTION TEST_CASE_2_EXEC:
                        IF vTestCases[1].state = utTestCaseStates.ut_RUNNING THEN
	(*Run the test case*)
	IF assertLessEqual_DWORD(vTestCase2_act, vTestCase2_xp) THEN
		vTestCases[1].state := utTestCaseStates.ut_PASSED;
		vTestCases[1].msg := 'Parameter act was equal to xp and function returned TRUE -> PASS';
	ELSE
		vTestCases[1].state := utTestCaseStates.ut_FAILED;
		vTestCases[1].msg := 'Parameter act was equal to xp and function returned FALSE -> FAIL';
	END_IF
END_IF
                      
END_ACTION

ACTION TEST_CASE_3_EXEC:
                        IF vTestCases[2].state = utTestCaseStates.ut_RUNNING THEN
	(*Run the test case*)
	IF NOT assertLessEqual_DWORD(vTestCase3_act, vTestCase3_xp) THEN
		vTestCases[2].state := utTestCaseStates.ut_PASSED;
		vTestCases[2].msg := 'Parameter act was greater than xp and function returned FALSE -> PASS';
	ELSE
		vTestCases[2].state := utTestCaseStates.ut_FAILED;
		vTestCases[2].msg := 'Parameter act was greater than xp and function returned TRUE -> FAIL';
	END_IF
END_IF
                      
END_ACTION

ACTION TEST_CASE_1_SETUP:
                        IF vTestCases[0].state = utTestCaseStates.ut_SETUP THEN
	(*Setup the test case information*)
	vTestCases[0].id := 1;
	vTestCases[0].desc[0] := 'RETURNS TRUE WHEN PARAMETER ACT LESS THAN XP';
    vTestCases[0].desc[1] := 'Tests if the function returns True if the parameter act is less than parameter xp';
	vTestCases[0].desc[2] := 'PASS IF: Return value is TRUE';
	
	(*Setup needed variables*)
	vTestCase1_act := REAL_TO_DWORD(85.4);
	vTestCase1_xp := REAL_TO_DWORD(115.4);
END_IF
                      
END_ACTION

ACTION TEST_CASE_1_EXEC:
                        IF vTestCases[0].state = utTestCaseStates.ut_RUNNING THEN
	(*Run the test case*)
	IF assertLessEqual_DWORD(vTestCase1_act, vTestCase1_xp) THEN
		vTestCases[0].state := utTestCaseStates.ut_PASSED;
		vTestCases[0].msg := 'Parameter act was less than xp and function returned TRUE -> PASS';
	ELSE
		vTestCases[0].state := utTestCaseStates.ut_FAILED;
		vTestCases[0].msg := 'Parameter act was less than xp and function returned FALSE -> FAIL';
	END_IF
END_IF
                      
END_ACTION

ACTION TEST_CASE_2_SETUP:
                        IF vTestCases[1].state = utTestCaseStates.ut_SETUP THEN
	(*Setup the test case information*)
	vTestCases[1].id := 2;
    vTestCases[1].desc[0] := 'RETURNS TRUE WHEN PARAMETER ACT EQUAL TO XP';
    vTestCases[1].desc[1] := 'Tests if the function returns True if the parameter act is equal to parameter xp';
	vTestCases[1].desc[2] := 'PASS IF: Return value is TRUE';
	
	(*Setup needed variables*)
	vTestCase2_act := REAL_TO_DWORD(115.4);
	vTestCase2_xp := REAL_TO_DWORD(115.4);
END_IF
                      
END_ACTION

ACTION TEST_CASE_3_SETUP:
                        IF vTestCases[2].state = utTestCaseStates.ut_SETUP THEN
	(*Setup the test case information*)
	vTestCases[2].id := 3;
    vTestCases[2].desc[0] := 'RETURNS FALSE WHEN PARAMETER ACT GREATER THAN XP';
    vTestCases[2].desc[1] := 'Tests if the function returns False if the parameter act is greater than parameter xp';
	vTestCases[2].desc[2] := 'PASS IF: Return value is FALSE';
	
	(*Setup needed variables*)
	vTestCase3_act := REAL_TO_DWORD(115.4);
	vTestCase3_xp := REAL_TO_DWORD(85.4);
END_IF
                      
END_ACTION
END_PROGRAM

PROGRAM test_assertLess_LWORD
  VAR
    vTestCases : ARRAY[0..20] OF utTestCase;  (* Definition of all test cases for this POU *)
    testRunner : utTestSuite;  (* Test Suite fb instance to run the tests *)
    vRunAll : BOOL;  (* Manual command to run all tests for this POU *)
    vResetAll : BOOL;  (* Manual command to reset all tests for this POU *)
    vTestCase1_act : LWORD;  (* Test data 1 of test case 1 *)
    vTestCase1_xp : LWORD;  (* Test data 2 of test case 1 *)
    vTestCase2_act : LWORD;  (* Test data 1 of test case 2 *)
    vTestCase2_xp : LWORD;  (* Test data 2 of test case 2 *)
  END_VAR

                    (*Run the test cases*)
TEST_CASE_1_SETUP();
TEST_CASE_1_EXEC();

TEST_CASE_2_SETUP();
TEST_CASE_2_EXEC();

(*Instantiate the test runner*)
testRunner(
	Id := 97,
	Name := 'assertLess_LWORD',
    RunTests := GVL.RunAll OR vRunAll,
	ResetTests := GVL.ResetAll OR vResetAll,
	TestCases:=vTestCases);

(*Report the results to the collection global*)
GVL.Results[testRunner.Id] := testRunner.Summary;
                  

ACTION TEST_CASE_2_EXEC:
                        IF vTestCases[1].state = utTestCaseStates.ut_RUNNING THEN
	(*Run the test case*)
	IF NOT assertLess_LWORD(vTestCase2_act, vTestCase2_xp) THEN
		vTestCases[1].state := utTestCaseStates.ut_PASSED;
		vTestCases[1].msg := 'Parameter act was greater than xp and function returned FALSE -> PASS';
	ELSE
		vTestCases[1].state := utTestCaseStates.ut_FAILED;
		vTestCases[1].msg := 'Parameter act was greater than xp and function returned TRUE -> FAIL';
	END_IF
END_IF
                      
END_ACTION

ACTION TEST_CASE_1_SETUP:
                        IF vTestCases[0].state = utTestCaseStates.ut_SETUP THEN
	(*Setup the test case information*)
	vTestCases[0].id := 1;
	vTestCases[0].desc[0] := 'RETURNS TRUE WHEN PARAMETER ACT LESS THAN XP';
    vTestCases[0].desc[1] := 'Tests if the function returns True if the parameter act is less than parameter xp';
	vTestCases[0].desc[2] := 'PASS IF: Return value is TRUE';
	
	(*Setup needed variables*)
	vTestCase1_act := REAL_TO_LWORD(85.4);
	vTestCase1_xp := REAL_TO_LWORD(115.4);
END_IF
                      
END_ACTION

ACTION TEST_CASE_1_EXEC:
                        IF vTestCases[0].state = utTestCaseStates.ut_RUNNING THEN
	(*Run the test case*)
	IF assertLess_LWORD(vTestCase1_act, vTestCase1_xp) THEN
		vTestCases[0].state := utTestCaseStates.ut_PASSED;
		vTestCases[0].msg := 'Parameter act was less than xp and function returned TRUE -> PASS';
	ELSE
		vTestCases[0].state := utTestCaseStates.ut_FAILED;
		vTestCases[0].msg := 'Parameter act was less than xp and function returned FALSE -> FAIL';
	END_IF
END_IF
                      
END_ACTION

ACTION TEST_CASE_2_SETUP:
                        IF vTestCases[1].state = utTestCaseStates.ut_SETUP THEN
	(*Setup the test case information*)
	vTestCases[1].id := 2;
    vTestCases[1].desc[0] := 'RETURNS FALSE WHEN PARAMETER ACT GREATER THAN XP';
    vTestCases[1].desc[1] := 'Tests if the function returns False if the parameter act is greater than parameter xp';
	vTestCases[1].desc[2] := 'PASS IF: Return value is FALSE';
	
	(*Setup needed variables*)
	vTestCase2_act := REAL_TO_LWORD(115.4);
	vTestCase2_xp := REAL_TO_LWORD(85.4);
END_IF
                      
END_ACTION
END_PROGRAM

PROGRAM test_assertLessEqual_WORD
  VAR
    vTestCases : ARRAY[0..20] OF utTestCase;  (* Definition of all test cases for this POU *)
    testRunner : utTestSuite;  (* Test Suite fb instance to run the tests *)
    vRunAll : BOOL;  (* Manual command to run all tests for this POU *)
    vResetAll : BOOL;  (* Manual command to reset all tests for this POU *)
    vTestCase1_act : WORD;  (* Test data 1 of test case 1 *)
    vTestCase1_xp : WORD;  (* Test data 2 of test case 1 *)
    vTestCase2_act : WORD;  (* Test data 1 of test case 2 *)
    vTestCase2_xp : WORD;  (* Test data 2 of test case 2 *)
    vTestCase3_act : WORD;  (* Test data 1 of test case 3 *)
    vTestCase3_xp : WORD;  (* Test data 2 of test case 3 *)
  END_VAR

                    (*Run the test cases*)
TEST_CASE_1_SETUP();
TEST_CASE_1_EXEC();

TEST_CASE_2_SETUP();
TEST_CASE_2_EXEC();

TEST_CASE_3_SETUP();
TEST_CASE_3_EXEC();

(*Instantiate the test runner*)
testRunner(
	Id := 117,
	Name := 'assertLessEqual_WORD',
    RunTests := GVL.RunAll OR vRunAll,
	ResetTests := GVL.ResetAll OR vResetAll,
	TestCases:=vTestCases);

(*Report the results to the collection global*)
GVL.Results[testRunner.Id] := testRunner.Summary;
                  

ACTION TEST_CASE_1_EXEC:
                        IF vTestCases[0].state = utTestCaseStates.ut_RUNNING THEN
	(*Run the test case*)
	IF assertLessEqual_WORD(vTestCase1_act, vTestCase1_xp) THEN
		vTestCases[0].state := utTestCaseStates.ut_PASSED;
		vTestCases[0].msg := 'Parameter act was less than xp and function returned TRUE -> PASS';
	ELSE
		vTestCases[0].state := utTestCaseStates.ut_FAILED;
		vTestCases[0].msg := 'Parameter act was less than xp and function returned FALSE -> FAIL';
	END_IF
END_IF
                      
END_ACTION

ACTION TEST_CASE_2_SETUP:
                        IF vTestCases[1].state = utTestCaseStates.ut_SETUP THEN
	(*Setup the test case information*)
	vTestCases[1].id := 2;
    vTestCases[1].desc[0] := 'RETURNS TRUE WHEN PARAMETER ACT EQUAL TO XP';
    vTestCases[1].desc[1] := 'Tests if the function returns True if the parameter act is equal to parameter xp';
	vTestCases[1].desc[2] := 'PASS IF: Return value is TRUE';
	
	(*Setup needed variables*)
	vTestCase2_act := REAL_TO_WORD(115.4);
	vTestCase2_xp := REAL_TO_WORD(115.4);
END_IF
                      
END_ACTION

ACTION TEST_CASE_2_EXEC:
                        IF vTestCases[1].state = utTestCaseStates.ut_RUNNING THEN
	(*Run the test case*)
	IF assertLessEqual_WORD(vTestCase2_act, vTestCase2_xp) THEN
		vTestCases[1].state := utTestCaseStates.ut_PASSED;
		vTestCases[1].msg := 'Parameter act was equal to xp and function returned TRUE -> PASS';
	ELSE
		vTestCases[1].state := utTestCaseStates.ut_FAILED;
		vTestCases[1].msg := 'Parameter act was equal to xp and function returned FALSE -> FAIL';
	END_IF
END_IF
                      
END_ACTION

ACTION TEST_CASE_1_SETUP:
                        IF vTestCases[0].state = utTestCaseStates.ut_SETUP THEN
	(*Setup the test case information*)
	vTestCases[0].id := 1;
	vTestCases[0].desc[0] := 'RETURNS TRUE WHEN PARAMETER ACT LESS THAN XP';
    vTestCases[0].desc[1] := 'Tests if the function returns True if the parameter act is less than parameter xp';
	vTestCases[0].desc[2] := 'PASS IF: Return value is TRUE';
	
	(*Setup needed variables*)
	vTestCase1_act := REAL_TO_WORD(85.4);
	vTestCase1_xp := REAL_TO_WORD(115.4);
END_IF
                      
END_ACTION

ACTION TEST_CASE_3_SETUP:
                        IF vTestCases[2].state = utTestCaseStates.ut_SETUP THEN
	(*Setup the test case information*)
	vTestCases[2].id := 3;
    vTestCases[2].desc[0] := 'RETURNS FALSE WHEN PARAMETER ACT GREATER THAN XP';
    vTestCases[2].desc[1] := 'Tests if the function returns False if the parameter act is greater than parameter xp';
	vTestCases[2].desc[2] := 'PASS IF: Return value is FALSE';
	
	(*Setup needed variables*)
	vTestCase3_act := REAL_TO_WORD(115.4);
	vTestCase3_xp := REAL_TO_WORD(85.4);
END_IF
                      
END_ACTION

ACTION TEST_CASE_3_EXEC:
                        IF vTestCases[2].state = utTestCaseStates.ut_RUNNING THEN
	(*Run the test case*)
	IF NOT assertLessEqual_WORD(vTestCase3_act, vTestCase3_xp) THEN
		vTestCases[2].state := utTestCaseStates.ut_PASSED;
		vTestCases[2].msg := 'Parameter act was greater than xp and function returned FALSE -> PASS';
	ELSE
		vTestCases[2].state := utTestCaseStates.ut_FAILED;
		vTestCases[2].msg := 'Parameter act was greater than xp and function returned TRUE -> FAIL';
	END_IF
END_IF
                      
END_ACTION
END_PROGRAM

PROGRAM test_assertLess_LINT
  VAR
    vTestCases : ARRAY[0..20] OF utTestCase;  (* Definition of all test cases for this POU *)
    testRunner : utTestSuite;  (* Test Suite fb instance to run the tests *)
    vRunAll : BOOL;  (* Manual command to run all tests for this POU *)
    vResetAll : BOOL;  (* Manual command to reset all tests for this POU *)
    vTestCase1_act : LINT;  (* Test data 1 of test case 1 *)
    vTestCase1_xp : LINT;  (* Test data 2 of test case 1 *)
    vTestCase2_act : LINT;  (* Test data 1 of test case 2 *)
    vTestCase2_xp : LINT;  (* Test data 2 of test case 2 *)
  END_VAR

                    (*Run the test cases*)
TEST_CASE_1_SETUP();
TEST_CASE_1_EXEC();

TEST_CASE_2_SETUP();
TEST_CASE_2_EXEC();

(*Instantiate the test runner*)
testRunner(
	Id := 104,
	Name := 'assertLess_LINT',
    RunTests := GVL.RunAll OR vRunAll,
	ResetTests := GVL.ResetAll OR vResetAll,
	TestCases:=vTestCases);

(*Report the results to the collection global*)
GVL.Results[testRunner.Id] := testRunner.Summary;
                  

ACTION TEST_CASE_2_EXEC:
                        IF vTestCases[1].state = utTestCaseStates.ut_RUNNING THEN
	(*Run the test case*)
	IF NOT assertLess_LINT(vTestCase2_act, vTestCase2_xp) THEN
		vTestCases[1].state := utTestCaseStates.ut_PASSED;
		vTestCases[1].msg := 'Parameter act was greater than xp and function returned FALSE -> PASS';
	ELSE
		vTestCases[1].state := utTestCaseStates.ut_FAILED;
		vTestCases[1].msg := 'Parameter act was greater than xp and function returned TRUE -> FAIL';
	END_IF
END_IF
                      
END_ACTION

ACTION TEST_CASE_1_SETUP:
                        IF vTestCases[0].state = utTestCaseStates.ut_SETUP THEN
	(*Setup the test case information*)
	vTestCases[0].id := 1;
	vTestCases[0].desc[0] := 'RETURNS TRUE WHEN PARAMETER ACT LESS THAN XP';
    vTestCases[0].desc[1] := 'Tests if the function returns True if the parameter act is less than parameter xp';
	vTestCases[0].desc[2] := 'PASS IF: Return value is TRUE';
	
	(*Setup needed variables*)
	vTestCase1_act := REAL_TO_LINT(85.4);
	vTestCase1_xp := REAL_TO_LINT(115.4);
END_IF
                      
END_ACTION

ACTION TEST_CASE_1_EXEC:
                        IF vTestCases[0].state = utTestCaseStates.ut_RUNNING THEN
	(*Run the test case*)
	IF assertLess_LINT(vTestCase1_act, vTestCase1_xp) THEN
		vTestCases[0].state := utTestCaseStates.ut_PASSED;
		vTestCases[0].msg := 'Parameter act was less than xp and function returned TRUE -> PASS';
	ELSE
		vTestCases[0].state := utTestCaseStates.ut_FAILED;
		vTestCases[0].msg := 'Parameter act was less than xp and function returned FALSE -> FAIL';
	END_IF
END_IF
                      
END_ACTION

ACTION TEST_CASE_2_SETUP:
                        IF vTestCases[1].state = utTestCaseStates.ut_SETUP THEN
	(*Setup the test case information*)
	vTestCases[1].id := 2;
    vTestCases[1].desc[0] := 'RETURNS FALSE WHEN PARAMETER ACT GREATER THAN XP';
    vTestCases[1].desc[1] := 'Tests if the function returns False if the parameter act is greater than parameter xp';
	vTestCases[1].desc[2] := 'PASS IF: Return value is FALSE';
	
	(*Setup needed variables*)
	vTestCase2_act := REAL_TO_LINT(115.4);
	vTestCase2_xp := REAL_TO_LINT(85.4);
END_IF
                      
END_ACTION
END_PROGRAM

PROGRAM test_assertLessEqual_LWORD
  VAR
    vTestCases : ARRAY[0..20] OF utTestCase;  (* Definition of all test cases for this POU *)
    testRunner : utTestSuite;  (* Test Suite fb instance to run the tests *)
    vRunAll : BOOL;  (* Manual command to run all tests for this POU *)
    vResetAll : BOOL;  (* Manual command to reset all tests for this POU *)
    vTestCase1_act : LWORD;  (* Test data 1 of test case 1 *)
    vTestCase1_xp : LWORD;  (* Test data 2 of test case 1 *)
    vTestCase2_act : LWORD;  (* Test data 1 of test case 2 *)
    vTestCase2_xp : LWORD;  (* Test data 2 of test case 2 *)
    vTestCase3_act : LWORD;  (* Test data 1 of test case 3 *)
    vTestCase3_xp : LWORD;  (* Test data 2 of test case 3 *)
  END_VAR

                    (*Run the test cases*)
TEST_CASE_1_SETUP();
TEST_CASE_1_EXEC();

TEST_CASE_2_SETUP();
TEST_CASE_2_EXEC();

TEST_CASE_3_SETUP();
TEST_CASE_3_EXEC();

(*Instantiate the test runner*)
testRunner(
	Id := 119,
	Name := 'assertLessEqual_LWORD',
    RunTests := GVL.RunAll OR vRunAll,
	ResetTests := GVL.ResetAll OR vResetAll,
	TestCases:=vTestCases);

(*Report the results to the collection global*)
GVL.Results[testRunner.Id] := testRunner.Summary;
                  

ACTION TEST_CASE_1_SETUP:
                        IF vTestCases[0].state = utTestCaseStates.ut_SETUP THEN
	(*Setup the test case information*)
	vTestCases[0].id := 1;
	vTestCases[0].desc[0] := 'RETURNS TRUE WHEN PARAMETER ACT LESS THAN XP';
    vTestCases[0].desc[1] := 'Tests if the function returns True if the parameter act is less than parameter xp';
	vTestCases[0].desc[2] := 'PASS IF: Return value is TRUE';
	
	(*Setup needed variables*)
	vTestCase1_act := REAL_TO_LWORD(85.4);
	vTestCase1_xp := REAL_TO_LWORD(115.4);
END_IF
                      
END_ACTION

ACTION TEST_CASE_1_EXEC:
                        IF vTestCases[0].state = utTestCaseStates.ut_RUNNING THEN
	(*Run the test case*)
	IF assertLessEqual_LWORD(vTestCase1_act, vTestCase1_xp) THEN
		vTestCases[0].state := utTestCaseStates.ut_PASSED;
		vTestCases[0].msg := 'Parameter act was less than xp and function returned TRUE -> PASS';
	ELSE
		vTestCases[0].state := utTestCaseStates.ut_FAILED;
		vTestCases[0].msg := 'Parameter act was less than xp and function returned FALSE -> FAIL';
	END_IF
END_IF
                      
END_ACTION

ACTION TEST_CASE_2_SETUP:
                        IF vTestCases[1].state = utTestCaseStates.ut_SETUP THEN
	(*Setup the test case information*)
	vTestCases[1].id := 2;
    vTestCases[1].desc[0] := 'RETURNS TRUE WHEN PARAMETER ACT EQUAL TO XP';
    vTestCases[1].desc[1] := 'Tests if the function returns True if the parameter act is equal to parameter xp';
	vTestCases[1].desc[2] := 'PASS IF: Return value is TRUE';
	
	(*Setup needed variables*)
	vTestCase2_act := REAL_TO_LWORD(115.4);
	vTestCase2_xp := REAL_TO_LWORD(115.4);
END_IF
                      
END_ACTION

ACTION TEST_CASE_2_EXEC:
                        IF vTestCases[1].state = utTestCaseStates.ut_RUNNING THEN
	(*Run the test case*)
	IF assertLessEqual_LWORD(vTestCase2_act, vTestCase2_xp) THEN
		vTestCases[1].state := utTestCaseStates.ut_PASSED;
		vTestCases[1].msg := 'Parameter act was equal to xp and function returned TRUE -> PASS';
	ELSE
		vTestCases[1].state := utTestCaseStates.ut_FAILED;
		vTestCases[1].msg := 'Parameter act was equal to xp and function returned FALSE -> FAIL';
	END_IF
END_IF
                      
END_ACTION

ACTION TEST_CASE_3_SETUP:
                        IF vTestCases[2].state = utTestCaseStates.ut_SETUP THEN
	(*Setup the test case information*)
	vTestCases[2].id := 3;
    vTestCases[2].desc[0] := 'RETURNS FALSE WHEN PARAMETER ACT GREATER THAN XP';
    vTestCases[2].desc[1] := 'Tests if the function returns False if the parameter act is greater than parameter xp';
	vTestCases[2].desc[2] := 'PASS IF: Return value is FALSE';
	
	(*Setup needed variables*)
	vTestCase3_act := REAL_TO_LWORD(115.4);
	vTestCase3_xp := REAL_TO_LWORD(85.4);
END_IF
                      
END_ACTION

